gfCNCPoint4[4846] = {X 266.6262, Y 56.8093, Z -5.5000, A 0.000, B 0.000, C 0.000 }
gfCNCPoint4[4847] = {X 266.8456, Y 55.6367, Z -5.5000, A 0.000, B 0.000, C 0.000 }
gfCNCPoint4[4848] = {X 267.2076, Y 54.5000, Z -5.5000, A 0.000, B 0.000, C 0.000 }
gfCNCPoint4[4849] = {X 267.7067, Y 53.4164, Z -5.5000, A 0.000, B 0.000, C 0.000 }
gfCNCPoint4[4850] = {X 268.4728, Y 52.2132, Z -5.5000, A 0.000, B 0.000, C 0.000 }
gfCNCPoint4[4851] = {X 269.4075, Y 51.1357, Z -5.5000, A 0.000, B 0.000, C 0.000 }
gfCNCPoint4[4852] = {X 270.4903, Y 50.2072, Z -5.5000, A 0.000, B 0.000, C 0.000 }
gfCNCPoint4[4853] = {X 271.6979, Y 49.4479, Z -5.5000, A 0.000, B 0.000, C 0.000 }
gfCNCPoint4[4854] = {X 273.0039, Y 48.8744, Z -5.5000, A 0.000, B 0.000, C 0.000 }
gfCNCPoint4[4855] = {X 274.3800, Y 48.4989, Z -5.5000, A 0.000, B 0.000, C 0.000 }
gfCNCPoint4[4856] = {X 275.3020, Y 48.3648, Z -5.5000, A 0.000, B 0.000, C 0.000 }
gfCNCPoint4[4857] = {X 276.2327, Y 48.3200, Z -5.5000, A 0.000, B 0.000, C 0.000 }
gfCNCPoint4[4858] = {X 281.0411, Y 48.3200, Z -5.5000, A 0.000, B 0.000, C 0.000 }
gfCNCPoint4[4859] = {X 280.4347, Y 47.5134, Z -5.5000, A 0.000, B 0.000, C 0.000 }
gfCNCPoint4[4860] = {X 280.0072, Y 46.5992, Z -5.5000, A 0.000, B 0.000, C 0.000 }
gfCNCPoint4[4861] = {X 279.7768, Y 45.6167, Z -5.5000, A 0.000, B 0.000, C 0.000 }
gfCNCPoint4[4862] = {X 279.7488, Y 45.3288, Z -5.5000, A 0.000, B 0.000, C 0.000 }
gfCNCPoint4[4863] = {X 279.7378, Y 45.0398, Z -5.5000, A 0.000, B 0.000, C 0.000 }
gfCNCPoint4[4864] = {X 279.7377, Y 44.2045, Z -5.5000, A 0.000, B 0.000, C 0.000 }
gfCNCPoint4[4865] = {X 279.8418, Y 43.2208, Z -5.5000, A 0.000, B 0.000, C 0.000 }
gfCNCPoint4[4866] = {X 280.1403, Y 42.2777, Z -5.5000, A 0.000, B 0.000, C 0.000 }
gfCNCPoint4[4867] = {X 280.6212, Y 41.4133, Z -5.5000, A 0.000, B 0.000, C 0.000 }
gfCNCPoint4[4868] = {X 281.2650, Y 40.6623, Z -5.5000, A 0.000, B 0.000, C 0.000 }
gfCNCPoint4[4869] = {X 281.2646, Y 16.5236, Z -5.5000, A 0.000, B 0.000, C 0.000 }
gfCNCPoint4[4870] = {X 280.6237, Y 15.7821, Z -5.5000, A 0.000, B 0.000, C 0.000 }
gfCNCPoint4[4871] = {X 280.1439, Y 14.9274, Z -5.5000, A 0.000, B 0.000, C 0.000 }
gfCNCPoint4[4872] = {X 279.8446, Y 13.9941, Z -5.5000, A 0.000, B 0.000, C 0.000 }
gfCNCPoint4[4873] = {X 279.7378, Y 13.0198, Z -5.5000, A 0.000, B 0.000, C 0.000 }
gfCNCPoint4[4874] = {X 279.7377, Y 12.1868, Z -5.5000, A 0.000, B 0.000, C 0.000 }
gfCNCPoint4[4875] = {X 279.8242, Y 11.2717, Z -5.5000, A 0.000, B 0.000, C 0.000 }
gfCNCPoint4[4876] = {X 280.0809, Y 10.3891, Z -5.5000, A 0.000, B 0.000, C 0.000 }
gfCNCPoint4[4877] = {X 280.5256, Y 9.5280, Z -5.5000, A 0.000, B 0.000, C 0.000 }
gfCNCPoint4[4878] = {X 281.1317, Y 8.7718, Z -5.5000, A 0.000, B 0.000, C 0.000 }
gfCNCPoint4[4879] = {X 281.8753, Y 8.1503, Z -5.5000, A 0.000, B 0.000, C 0.000 }
gfCNCPoint4[4880] = {X 282.7270, Y 7.6879, Z -5.5000, A 0.000, B 0.000, C 0.000 }
gfCNCPoint4[4881] = {X 283.6533, Y 7.4030, Z -5.5000, A 0.000, B 0.000, C 0.000 }
gfCNCPoint4[4882] = {X 284.6177, Y 7.3068, Z -5.5000, A 0.000, B 0.000, C 0.000 }
gfCNCPoint4[4883] = {X 291.0611, Y 7.3068, Z -5.5000, A 0.000, B 0.000, C 0.000 }
gfCNCPoint4[4884] = {X 292.0255, Y 7.4030, Z -5.5000, A 0.000, B 0.000, C 0.000 }
gfCNCPoint4[4885] = {X 292.9518, Y 7.6879, Z -5.5000, A 0.000, B 0.000, C 0.000 }
gfCNCPoint4[4886] = {X 293.8035, Y 8.1503, Z -5.5000, A 0.000, B 0.000, C 0.000 }
gfCNCPoint4[4887] = {X 294.5471, Y 8.7718, Z -5.5000, A 0.000, B 0.000, C 0.000 }
gfCNCPoint4[4888] = {X 295.1532, Y 9.5280, Z -5.5000, A 0.000, B 0.000, C 0.000 }
gfCNCPoint4[4889] = {X 295.5979, Y 10.3891, Z -5.5000, A 0.000, B 0.000, C 0.000 }
gfCNCPoint4[4890] = {X 295.8044, Y 11.0397, Z -5.5000, A 0.000, B 0.000, C 0.000 }
gfCNCPoint4[4891] = {X 295.9180, Y 11.7127, Z -5.5000, A 0.000, B 0.000, C 0.000 }
gfCNCPoint4[4892] = {X 295.9354, Y 11.9495, Z -5.5000, A 0.000, B 0.000, C 0.000 }
gfCNCPoint4[4893] = {X 295.9411, Y 12.1868, Z -5.5000, A 0.000, B 0.000, C 0.000 }
gfCNCPoint4[4894] = {X 295.9409, Y 13.0237, Z -5.5000, A 0.000, B 0.000, C 0.000 }
gfCNCPoint4[4895] = {X 295.9342, Y 13.2382, Z -5.5000, A 0.000, B 0.000, C 0.000 }
gfCNCPoint4[4896] = {X 295.9180, Y 13.4521, Z -5.5000, A 0.000, B 0.000, C 0.000 }
gfCNCPoint4[4897] = {X 298.3067, Y 13.6853, Z -5.5000, A 0.000, B 0.000, C 0.000 }
gfCNCPoint4[4898] = {X 298.1361, Y 14.6935, Z -5.5000, A 0.000, B 0.000, C 0.000 }
gfCNCPoint4[4899] = {X 297.8260, Y 15.6678, Z -5.5000, A 0.000, B 0.000, C 0.000 }
gfCNCPoint4[4900] = {X 297.3824, Y 16.5891, Z -5.5000, A 0.000, B 0.000, C 0.000 }
gfCNCPoint4[4901] = {X 296.8141, Y 17.4392, Z -5.5000, A 0.000, B 0.000, C 0.000 }
gfCNCPoint4[4902] = {X 296.8144, Y 19.2365, Z -5.5000, A 0.000, B 0.000, C 0.000 }
gfCNCPoint4[4903] = {X 299.7989, Y 19.2365, Z -5.5000, A 0.000, B 0.000, C 0.000 }
gfCNCPoint4[4904] = {X 299.7990, Y 17.4388, Z -5.5000, A 0.000, B 0.000, C 0.000 }
gfCNCPoint4[4905] = {X 299.2308, Y 16.5888, Z -5.5000, A 0.000, B 0.000, C 0.000 }
gfCNCPoint4[4906] = {X 298.7873, Y 15.6676, Z -5.5000, A 0.000, B 0.000, C 0.000 }
gfCNCPoint4[4907] = {X 298.4772, Y 14.6934, Z -5.5000, A 0.000, B 0.000, C 0.000 }
gfCNCPoint4[4908] = {X 298.3067, Y 13.6853, Z -5.5000, A 0.000, B 0.000, C 0.000 }
gfCNCPoint4[4909] = {X 295.9180, Y 13.4521, Z -5.5000, A 0.000, B 0.000, C 0.000 }
gfCNCPoint4[4910] = {X 295.7560, Y 14.3094, Z -5.5000, A 0.000, B 0.000, C 0.000 }
gfCNCPoint4[4911] = {X 295.4439, Y 15.1241, Z -5.5000, A 0.000, B 0.000, C 0.000 }
gfCNCPoint4[4912] = {X 294.9917, Y 15.8702, Z -5.5000, A 0.000, B 0.000, C 0.000 }
gfCNCPoint4[4913] = {X 294.4139, Y 16.5239, Z -5.5000, A 0.000, B 0.000, C 0.000 }
gfCNCPoint4[4914] = {X 294.4148, Y 21.6365, Z -5.5000, A 0.000, B 0.000, C 0.000 }
gfCNCPoint4[4915] = {X 302.1988, Y 21.6365, Z -5.5000, A 0.000, B 0.000, C 0.000 }
gfCNCPoint4[4916] = {X 302.1991, Y 16.5235, Z -5.5000, A 0.000, B 0.000, C 0.000 }
gfCNCPoint4[4917] = {X 301.6214, Y 15.8699, Z -5.5000, A 0.000, B 0.000, C 0.000 }
gfCNCPoint4[4918] = {X 301.1694, Y 15.1239, Z -5.5000, A 0.000, B 0.000, C 0.000 }
gfCNCPoint4[4919] = {X 300.8573, Y 14.3093, Z -5.5000, A 0.000, B 0.000, C 0.000 }
gfCNCPoint4[4920] = {X 300.6953, Y 13.4521, Z -5.5000, A 0.000, B 0.000, C 0.000 }
gfCNCPoint4[4921] = {X 300.6791, Y 13.2371, Z -5.5000, A 0.000, B 0.000, C 0.000 }
gfCNCPoint4[4922] = {X 300.6724, Y 13.0215, Z -5.5000, A 0.000, B 0.000, C 0.000 }
gfCNCPoint4[4923] = {X 300.6723, Y 12.1868, Z -5.5000, A 0.000, B 0.000, C 0.000 }
gfCNCPoint4[4924] = {X 300.6780, Y 11.9495, Z -5.5000, A 0.000, B 0.000, C 0.000 }
gfCNCPoint4[4925] = {X 300.6953, Y 11.7127, Z -5.5000, A 0.000, B 0.000, C 0.000 }
gfCNCPoint4[4926] = {X 300.8090, Y 11.0397, Z -5.5000, A 0.000, B 0.000, C 0.000 }
gfCNCPoint4[4927] = {X 301.0155, Y 10.3891, Z -5.5000, A 0.000, B 0.000, C 0.000 }
gfCNCPoint4[4928] = {X 301.4602, Y 9.5280, Z -5.5000, A 0.000, B 0.000, C 0.000 }
gfCNCPoint4[4929] = {X 302.0663, Y 8.7718, Z -5.5000, A 0.000, B 0.000, C 0.000 }
gfCNCPoint4[4930] = {X 302.8099, Y 8.1503, Z -5.5000, A 0.000, B 0.000, C 0.000 }
gfCNCPoint4[4931] = {X 303.6616, Y 7.6879, Z -5.5000, A 0.000, B 0.000, C 0.000 }
gfCNCPoint4[4932] = {X 304.5879, Y 7.4030, Z -5.5000, A 0.000, B 0.000, C 0.000 }
gfCNCPoint4[4933] = {X 305.5523, Y 7.3068, Z -5.5000, A 0.000, B 0.000, C 0.000 }
gfCNCPoint4[4934] = {X 311.9957, Y 7.3068, Z -5.5000, A 0.000, B 0.000, C 0.000 }
gfCNCPoint4[4935] = {X 312.9478, Y 7.4006, Z -5.5000, A 0.000, B 0.000, C 0.000 }
gfCNCPoint4[4936] = {X 313.8632, Y 7.6783, Z -5.5000, A 0.000, B 0.000, C 0.000 }
gfCNCPoint4[4937] = {X 314.7069, Y 8.1292, Z -5.5000, A 0.000, B 0.000, C 0.000 }
gfCNCPoint4[4938] = {X 315.4464, Y 8.7361, Z -5.5000, A 0.000, B 0.000, C 0.000 }
gfCNCPoint4[4939] = {X 316.0533, Y 9.4756, Z -5.5000, A 0.000, B 0.000, C 0.000 }
gfCNCPoint4[4940] = {X 316.5043, Y 10.3193, Z -5.5000, A 0.000, B 0.000, C 0.000 }
gfCNCPoint4[4941] = {X 316.7820, Y 11.2348, Z -5.5000, A 0.000, B 0.000, C 0.000 }
gfCNCPoint4[4942] = {X 316.8757, Y 12.1868, Z -5.5000, A 0.000, B 0.000, C 0.000 }
gfCNCPoint4[4943] = {X 316.8755, Y 13.0237, Z -5.5000, A 0.000, B 0.000, C 0.000 }
gfCNCPoint4[4944] = {X 316.7682, Y 13.9967, Z -5.5000, A 0.000, B 0.000, C 0.000 }
gfCNCPoint4[4945] = {X 316.4689, Y 14.9287, Z -5.5000, A 0.000, B 0.000, C 0.000 }
gfCNCPoint4[4946] = {X 315.9895, Y 15.7823, Z -5.5000, A 0.000, B 0.000, C 0.000 }
gfCNCPoint4[4947] = {X 315.3495, Y 16.5229, Z -5.5000, A 0.000, B 0.000, C 0.000 }
gfCNCPoint4[4948] = {X 315.3484, Y 40.6628, Z -5.5000, A 0.000, B 0.000, C 0.000 }
gfCNCPoint4[4949] = {X 315.9894, Y 41.4043, Z -5.5000, A 0.000, B 0.000, C 0.000 }
gfCNCPoint4[4950] = {X 316.4692, Y 42.2589, Z -5.5000, A 0.000, B 0.000, C 0.000 }
gfCNCPoint4[4951] = {X 316.7687, Y 43.1922, Z -5.5000, A 0.000, B 0.000, C 0.000 }
gfCNCPoint4[4952] = {X 316.8755, Y 44.1664, Z -5.5000, A 0.000, B 0.000, C 0.000 }
gfCNCPoint4[4953] = {X 316.8757, Y 45.0000, Z -5.5000, A 0.000, B 0.000, C 0.000 }
gfCNCPoint4[4954] = {X 316.8749, Y 45.0899, Z -5.5000, A 0.000, B 0.000, C 0.000 }
gfCNCPoint4[4955] = {X 316.8724, Y 45.1799, Z -5.5000, A 0.000, B 0.000, C 0.000 }
gfCNCPoint4[4956] = {X 316.8594, Y 45.3987, Z -5.5000, A 0.000, B 0.000, C 0.000 }
gfCNCPoint4[4957] = {X 316.8366, Y 45.6167, Z -5.5000, A 0.000, B 0.000, C 0.000 }
gfCNCPoint4[4958] = {X 316.6062, Y 46.5992, Z -5.5000, A 0.000, B 0.000, C 0.000 }
gfCNCPoint4[4959] = {X 316.1787, Y 47.5134, Z -5.5000, A 0.000, B 0.000, C 0.000 }
gfCNCPoint4[4960] = {X 315.5723, Y 48.3200, Z -5.5000, A 0.000, B 0.000, C 0.000 }
gfCNCPoint4[4961] = {X 315.2205, Y 47.9934, Z -5.5000, A 0.000, B 0.000, C 0.000 }
gfCNCPoint4[4962] = {X 314.5413, Y 48.5889, Z -5.5000, A 0.000, B 0.000, C 0.000 }
gfCNCPoint4[4963] = {X 313.7548, Y 49.0331, Z -5.5000, A 0.000, B 0.000, C 0.000 }
gfCNCPoint4[4964] = {X 312.8942, Y 49.3073, Z -5.5000, A 0.000, B 0.000, C 0.000 }
gfCNCPoint4[4965] = {X 311.9957, Y 49.4000, Z -5.5000, A 0.000, B 0.000, C 0.000 }
gfCNCPoint4[4966] = {X 305.5523, Y 49.4000, Z -5.5000, A 0.000, B 0.000, C 0.000 }
gfCNCPoint4[4967] = {X 304.5732, Y 49.2897, Z -5.5000, A 0.000, B 0.000, C 0.000 }
gfCNCPoint4[4968] = {X 303.6432, Y 48.9643, Z -5.5000, A 0.000, B 0.000, C 0.000 }
gfCNCPoint4[4969] = {X 302.8089, Y 48.4400, Z -5.5000, A 0.000, B 0.000, C 0.000 }
gfCNCPoint4[4970] = {X 302.1122, Y 47.7433, Z -5.5000, A 0.000, B 0.000, C 0.000 }
gfCNCPoint4[4971] = {X 301.5880, Y 46.9091, Z -5.5000, A 0.000, B 0.000, C 0.000 }
gfCNCPoint4[4972] = {X 301.2626, Y 45.9791, Z -5.5000, A 0.000, B 0.000, C 0.000 }
gfCNCPoint4[4973] = {X 301.1523, Y 45.0000, Z -5.5000, A 0.000, B 0.000, C 0.000 }
gfCNCPoint4[4974] = {X 301.1524, Y 44.1994, Z -5.5000, A 0.000, B 0.000, C 0.000 }
gfCNCPoint4[4975] = {X 301.2698, Y 43.2559, Z -5.5000, A 0.000, B 0.000, C 0.000 }
gfCNCPoint4[4976] = {X 301.5727, Y 42.3547, Z -5.5000, A 0.000, B 0.000, C 0.000 }
gfCNCPoint4[4977] = {X 302.0489, Y 41.5318, Z -5.5000, A 0.000, B 0.000, C 0.000 }
gfCNCPoint4[4978] = {X 302.6794, Y 40.8202, Z -5.5000, A 0.000, B 0.000, C 0.000 }
gfCNCPoint4[4979] = {X 302.6794, Y 34.1143, Z -5.5000, A 0.000, B 0.000, C 0.000 }
gfCNCPoint4[4980] = {X 293.9347, Y 34.1143, Z -5.5000, A 0.000, B 0.000, C 0.000 }
gfCNCPoint4[4981] = {X 293.9340, Y 40.8658, Z -5.5000, A 0.000, B 0.000, C 0.000 }
gfCNCPoint4[4982] = {X 294.5740, Y 41.5608, Z -5.5000, A 0.000, B 0.000, C 0.000 }
gfCNCPoint4[4983] = {X 295.0547, Y 42.3742, Z -5.5000, A 0.000, B 0.000, C 0.000 }
gfCNCPoint4[4984] = {X 295.3548, Y 43.2701, Z -5.5000, A 0.000, B 0.000, C 0.000 }
gfCNCPoint4[4985] = {X 295.4611, Y 44.2089, Z -5.5000, A 0.000, B 0.000, C 0.000 }
gfCNCPoint4[4986] = {X 295.4611, Y 45.0000, Z -5.5000, A 0.000, B 0.000, C 0.000 }
gfCNCPoint4[4987] = {X 295.3508, Y 45.9791, Z -5.5000, A 0.000, B 0.000, C 0.000 }
gfCNCPoint4[4988] = {X 295.0254, Y 46.9091, Z -5.5000, A 0.000, B 0.000, C 0.000 }
gfCNCPoint4[4989] = {X 294.5012, Y 47.7434, Z -5.5000, A 0.000, B 0.000, C 0.000 }
gfCNCPoint4[4990] = {X 293.8045, Y 48.4401, Z -5.5000, A 0.000, B 0.000, C 0.000 }
gfCNCPoint4[4991] = {X 292.9702, Y 48.9643, Z -5.5000, A 0.000, B 0.000, C 0.000 }
gfCNCPoint4[4992] = {X 292.0402, Y 49.2897, Z -5.5000, A 0.000, B 0.000, C 0.000 }
gfCNCPoint4[4993] = {X 291.0611, Y 49.4000, Z -5.5000, A 0.000, B 0.000, C 0.000 }
gfCNCPoint4[4994] = {X 284.6177, Y 49.4000, Z -5.5000, A 0.000, B 0.000, C 0.000 }
gfCNCPoint4[4995] = {X 283.6386, Y 49.2897, Z -5.5000, A 0.000, B 0.000, C 0.000 }
gfCNCPoint4[4996] = {X 282.7086, Y 48.9643, Z -5.5000, A 0.000, B 0.000, C 0.000 }
gfCNCPoint4[4997] = {X 281.8743, Y 48.4400, Z -5.5000, A 0.000, B 0.000, C 0.000 }
gfCNCPoint4[4998] = {X 281.1776, Y 47.7433, Z -5.5000, A 0.000, B 0.000, C 0.000 }
gfCNCPoint4[4999] = {X 280.6534, Y 46.9091, Z -5.5000, A 0.000, B 0.000, C 0.000 }
gfCNCPoint4[5000] = {X 280.3280, Y 45.9791, Z -5.5000, A 0.000, B 0.000, C 0.000 }
gfCNCPoint4[5001] = {X 280.2177, Y 45.0000, Z -5.5000, A 0.000, B 0.000, C 0.000 }
gfCNCPoint4[5002] = {X 280.2177, Y 44.2069, Z -5.5000, A 0.000, B 0.000, C 0.000 }
gfCNCPoint4[5003] = {X 280.3222, Y 43.2698, Z -5.5000, A 0.000, B 0.000, C 0.000 }
gfCNCPoint4[5004] = {X 280.6220, Y 42.3758, Z -5.5000, A 0.000, B 0.000, C 0.000 }
gfCNCPoint4[5005] = {X 281.1034, Y 41.5651, Z -5.5000, A 0.000, B 0.000, C 0.000 }
gfCNCPoint4[5006] = {X 281.7450, Y 40.8741, Z -5.5000, A 0.000, B 0.000, C 0.000 }
gfCNCPoint4[5007] = {X 281.7446, Y 16.3105, Z -5.5000, A 0.000, B 0.000, C 0.000 }
gfCNCPoint4[5008] = {X 281.1002, Y 15.6214, Z -5.5000, A 0.000, B 0.000, C 0.000 }
gfCNCPoint4[5009] = {X 280.6176, Y 14.8108, Z -5.5000, A 0.000, B 0.000, C 0.000 }
gfCNCPoint4[5010] = {X 280.3188, Y 13.9159, Z -5.5000, A 0.000, B 0.000, C 0.000 }
gfCNCPoint4[5011] = {X 280.2177, Y 12.9780, Z -5.5000, A 0.000, B 0.000, C 0.000 }
gfCNCPoint4[5012] = {X 280.2177, Y 12.1868, Z -5.5000, A 0.000, B 0.000, C 0.000 }
gfCNCPoint4[5013] = {X 280.3280, Y 11.2077, Z -5.5000, A 0.000, B 0.000, C 0.000 }
gfCNCPoint4[5014] = {X 280.6534, Y 10.2777, Z -5.5000, A 0.000, B 0.000, C 0.000 }
gfCNCPoint4[5015] = {X 281.1776, Y 9.4435, Z -5.5000, A 0.000, B 0.000, C 0.000 }
gfCNCPoint4[5016] = {X 281.8743, Y 8.7468, Z -5.5000, A 0.000, B 0.000, C 0.000 }
gfCNCPoint4[5017] = {X 282.7086, Y 8.2226, Z -5.5000, A 0.000, B 0.000, C 0.000 }
gfCNCPoint4[5018] = {X 283.6386, Y 7.8971, Z -5.5000, A 0.000, B 0.000, C 0.000 }
gfCNCPoint4[5019] = {X 284.6177, Y 7.7868, Z -5.5000, A 0.000, B 0.000, C 0.000 }
gfCNCPoint4[5020] = {X 291.0611, Y 7.7868, Z -5.5000, A 0.000, B 0.000, C 0.000 }
gfCNCPoint4[5021] = {X 292.0402, Y 7.8971, Z -5.5000, A 0.000, B 0.000, C 0.000 }
gfCNCPoint4[5022] = {X 292.9702, Y 8.2226, Z -5.5000, A 0.000, B 0.000, C 0.000 }
gfCNCPoint4[5023] = {X 293.8045, Y 8.7468, Z -5.5000, A 0.000, B 0.000, C 0.000 }
gfCNCPoint4[5024] = {X 294.5012, Y 9.4435, Z -5.5000, A 0.000, B 0.000, C 0.000 }
gfCNCPoint4[5025] = {X 295.0254, Y 10.2777, Z -5.5000, A 0.000, B 0.000, C 0.000 }
gfCNCPoint4[5026] = {X 295.3508, Y 11.2077, Z -5.5000, A 0.000, B 0.000, C 0.000 }
gfCNCPoint4[5027] = {X 295.4611, Y 12.1868, Z -5.5000, A 0.000, B 0.000, C 0.000 }
gfCNCPoint4[5028] = {X 295.4609, Y 13.0233, Z -5.5000, A 0.000, B 0.000, C 0.000 }
gfCNCPoint4[5029] = {X 295.3526, Y 13.9493, Z -5.5000, A 0.000, B 0.000, C 0.000 }
gfCNCPoint4[5030] = {X 295.0517, Y 14.8316, Z -5.5000, A 0.000, B 0.000, C 0.000 }
gfCNCPoint4[5031] = {X 294.5716, Y 15.6307, Z -5.5000, A 0.000, B 0.000, C 0.000 }
gfCNCPoint4[5032] = {X 293.9339, Y 16.3108, Z -5.5000, A 0.000, B 0.000, C 0.000 }
gfCNCPoint4[5033] = {X 293.9349, Y 22.1165, Z -5.5000, A 0.000, B 0.000, C 0.000 }
gfCNCPoint4[5034] = {X 302.6787, Y 22.1165, Z -5.5000, A 0.000, B 0.000, C 0.000 }
gfCNCPoint4[5035] = {X 302.6791, Y 16.3104, Z -5.5000, A 0.000, B 0.000, C 0.000 }
gfCNCPoint4[5036] = {X 302.0348, Y 15.6214, Z -5.5000, A 0.000, B 0.000, C 0.000 }
gfCNCPoint4[5037] = {X 301.5521, Y 14.8108, Z -5.5000, A 0.000, B 0.000, C 0.000 }
gfCNCPoint4[5038] = {X 301.2534, Y 13.9159, Z -5.5000, A 0.000, B 0.000, C 0.000 }
gfCNCPoint4[5039] = {X 301.1523, Y 12.9779, Z -5.5000, A 0.000, B 0.000, C 0.000 }
gfCNCPoint4[5040] = {X 301.1523, Y 12.1868, Z -5.5000, A 0.000, B 0.000, C 0.000 }
gfCNCPoint4[5041] = {X 301.2626, Y 11.2077, Z -5.5000, A 0.000, B 0.000, C 0.000 }
gfCNCPoint4[5042] = {X 301.5880, Y 10.2777, Z -5.5000, A 0.000, B 0.000, C 0.000 }
gfCNCPoint4[5043] = {X 302.1122, Y 9.4435, Z -5.5000, A 0.000, B 0.000, C 0.000 }
gfCNCPoint4[5044] = {X 302.8089, Y 8.7468, Z -5.5000, A 0.000, B 0.000, C 0.000 }
gfCNCPoint4[5045] = {X 303.6432, Y 8.2226, Z -5.5000, A 0.000, B 0.000, C 0.000 }
gfCNCPoint4[5046] = {X 304.5732, Y 7.8971, Z -5.5000, A 0.000, B 0.000, C 0.000 }
gfCNCPoint4[5047] = {X 305.5523, Y 7.7868, Z -5.5000, A 0.000, B 0.000, C 0.000 }
gfCNCPoint4[5048] = {X 311.9957, Y 7.7868, Z -5.5000, A 0.000, B 0.000, C 0.000 }
gfCNCPoint4[5049] = {X 312.9748, Y 7.8971, Z -5.5000, A 0.000, B 0.000, C 0.000 }
gfCNCPoint4[5050] = {X 313.9048, Y 8.2226, Z -5.5000, A 0.000, B 0.000, C 0.000 }
gfCNCPoint4[5051] = {X 314.7391, Y 8.7468, Z -5.5000, A 0.000, B 0.000, C 0.000 }
gfCNCPoint4[5052] = {X 315.4358, Y 9.4435, Z -5.5000, A 0.000, B 0.000, C 0.000 }
gfCNCPoint4[5053] = {X 315.9600, Y 10.2777, Z -5.5000, A 0.000, B 0.000, C 0.000 }
gfCNCPoint4[5054] = {X 316.2854, Y 11.2077, Z -5.5000, A 0.000, B 0.000, C 0.000 }
gfCNCPoint4[5055] = {X 316.3957, Y 12.1868, Z -5.5000, A 0.000, B 0.000, C 0.000 }
gfCNCPoint4[5056] = {X 316.3955, Y 13.0233, Z -5.5000, A 0.000, B 0.000, C 0.000 }
gfCNCPoint4[5057] = {X 316.2873, Y 13.9489, Z -5.5000, A 0.000, B 0.000, C 0.000 }
gfCNCPoint4[5058] = {X 315.9865, Y 14.8310, Z -5.5000, A 0.000, B 0.000, C 0.000 }
gfCNCPoint4[5059] = {X 315.5068, Y 15.6299, Z -5.5000, A 0.000, B 0.000, C 0.000 }
gfCNCPoint4[5060] = {X 314.8695, Y 16.3099, Z -5.5000, A 0.000, B 0.000, C 0.000 }
gfCNCPoint4[5061] = {X 314.8684, Y 40.8760, Z -5.5000, A 0.000, B 0.000, C 0.000 }
gfCNCPoint4[5062] = {X 315.5129, Y 41.5651, Z -5.5000, A 0.000, B 0.000, C 0.000 }
gfCNCPoint4[5063] = {X 315.9957, Y 42.3758, Z -5.5000, A 0.000, B 0.000, C 0.000 }
gfCNCPoint4[5064] = {X 316.2946, Y 43.2708, Z -5.5000, A 0.000, B 0.000, C 0.000 }
gfCNCPoint4[5065] = {X 316.3957, Y 44.2089, Z -5.5000, A 0.000, B 0.000, C 0.000 }
gfCNCPoint4[5066] = {X 316.3957, Y 45.0000, Z -5.5000, A 0.000, B 0.000, C 0.000 }
gfCNCPoint4[5067] = {X 316.3190, Y 45.8182, Z -5.5000, A 0.000, B 0.000, C 0.000 }
gfCNCPoint4[5068] = {X 316.0914, Y 46.6079, Z -5.5000, A 0.000, B 0.000, C 0.000 }
gfCNCPoint4[5069] = {X 315.7209, Y 47.3415, Z -5.5000, A 0.000, B 0.000, C 0.000 }
gfCNCPoint4[5070] = {X 315.2205, Y 47.9934, Z -5.5000, A 0.000, B 0.000, C 0.000 }
gfCNCPoint4[5071] = {X 315.5723, Y 48.3200, Z -5.5000, A 0.000, B 0.000, C 0.000 }
gfCNCPoint4[5072] = {X 324.3107, Y 48.3200, Z -5.5000, A 0.000, B 0.000, C 0.000 }
gfCNCPoint4[5073] = {X 325.5555, Y 48.4004, Z -5.5000, A 0.000, B 0.000, C 0.000 }
gfCNCPoint4[5074] = {X 326.7797, Y 48.6402, Z -5.5000, A 0.000, B 0.000, C 0.000 }
gfCNCPoint4[5075] = {X 325.5882, Y 48.0963, Z -5.5000, A 0.000, B 0.000, C 0.000 }
gfCNCPoint4[5076] = {X 324.4810, Y 47.3966, Z -5.5000, A 0.000, B 0.000, C 0.000 }
gfCNCPoint4[5077] = {X 323.4784, Y 46.5538, Z -5.5000, A 0.000, B 0.000, C 0.000 }
gfCNCPoint4[5078] = {X 322.8382, Y 45.9295, Z -5.5000, A 0.000, B 0.000, C 0.000 }
gfCNCPoint4[5079] = {X 322.2180, Y 45.2650, Z -5.5000, A 0.000, B 0.000, C 0.000 }
gfCNCPoint4[5080] = {X 321.6628, Y 44.5452, Z -5.5000, A 0.000, B 0.000, C 0.000 }
gfCNCPoint4[5081] = {X 323.6300, Y 43.1703, Z -5.5000, A 0.000, B 0.000, C 0.000 }
gfCNCPoint4[5082] = {X 323.0063, Y 42.0918, Z -5.5000, A 0.000, B 0.000, C 0.000 }
gfCNCPoint4[5083] = {X 322.5757, Y 40.9227, Z -5.5000, A 0.000, B 0.000, C 0.000 }
gfCNCPoint4[5084] = {X 322.3506, Y 39.6973, Z -5.5000, A 0.000, B 0.000, C 0.000 }
gfCNCPoint4[5085] = {X 322.3379, Y 38.4514, Z -5.5000, A 0.000, B 0.000, C 0.000 }
gfCNCPoint4[5086] = {X 322.5377, Y 37.2217, Z -5.5000, A 0.000, B 0.000, C 0.000 }
gfCNCPoint4[5087] = {X 322.9443, Y 36.0440, Z -5.5000, A 0.000, B 0.000, C 0.000 }
gfCNCPoint4[5088] = {X 323.5458, Y 34.9529, Z -5.5000, A 0.000, B 0.000, C 0.000 }
gfCNCPoint4[5089] = {X 327.7840, Y 28.6158, Z -5.5000, A 0.000, B 0.000, C 0.000 }
gfCNCPoint4[5090] = {X 328.5200, Y 27.6906, Z -5.5000, A 0.000, B 0.000, C 0.000 }
gfCNCPoint4[5091] = {X 329.3960, Y 26.8968, Z -5.5000, A 0.000, B 0.000, C 0.000 }
gfCNCPoint4[5092] = {X 330.3889, Y 26.2552, Z -5.5000, A 0.000, B 0.000, C 0.000 }
gfCNCPoint4[5093] = {X 331.5063, Y 25.7713, Z -5.5000, A 0.000, B 0.000, C 0.000 }
gfCNCPoint4[5094] = {X 332.6887, Y 25.4804, Z -5.5000, A 0.000, B 0.000, C 0.000 }
gfCNCPoint4[5095] = {X 333.9031, Y 25.3907, Z -5.5000, A 0.000, B 0.000, C 0.000 }
gfCNCPoint4[5096] = {X 335.1154, Y 25.5046, Z -5.5000, A 0.000, B 0.000, C 0.000 }
gfCNCPoint4[5097] = {X 336.2918, Y 25.8191, Z -5.5000, A 0.000, B 0.000, C 0.000 }
gfCNCPoint4[5098] = {X 337.3993, Y 26.3252, Z -5.5000, A 0.000, B 0.000, C 0.000 }
gfCNCPoint4[5099] = {X 338.1754, Y 26.8291, Z -5.5000, A 0.000, B 0.000, C 0.000 }
gfCNCPoint4[5100] = {X 338.8812, Y 27.4275, Z -5.5000, A 0.000, B 0.000, C 0.000 }
gfCNCPoint4[5101] = {X 339.5029, Y 28.0268, Z -5.5000, A 0.000, B 0.000, C 0.000 }
gfCNCPoint4[5102] = {X 340.3307, Y 28.9967, Z -5.5000, A 0.000, B 0.000, C 0.000 }
gfCNCPoint4[5103] = {X 340.9766, Y 30.0961, Z -5.5000, A 0.000, B 0.000, C 0.000 }
gfCNCPoint4[5104] = {X 341.4207, Y 31.2913, Z -5.5000, A 0.000, B 0.000, C 0.000 }
gfCNCPoint4[5105] = {X 341.6495, Y 32.5458, Z -5.5000, A 0.000, B 0.000, C 0.000 }
gfCNCPoint4[5106] = {X 341.8492, Y 32.7096, Z -5.5000, A 0.000, B 0.000, C 0.000 }
gfCNCPoint4[5107] = {X 342.0509, Y 32.8710, Z -5.5000, A 0.000, B 0.000, C 0.000 }
gfCNCPoint4[5108] = {X 342.9928, Y 33.4854, Z -5.5000, A 0.000, B 0.000, C 0.000 }
gfCNCPoint4[5109] = {X 344.0146, Y 33.9553, Z -5.5000, A 0.000, B 0.000, C 0.000 }
gfCNCPoint4[5110] = {X 345.0942, Y 34.2706, Z -5.5000, A 0.000, B 0.000, C 0.000 }
gfCNCPoint4[5111] = {X 346.2082, Y 34.4244, Z -5.5000, A 0.000, B 0.000, C 0.000 }
gfCNCPoint4[5112] = {X 347.3328, Y 34.4134, Z -5.5000, A 0.000, B 0.000, C 0.000 }
gfCNCPoint4[5113] = {X 348.3024, Y 34.2880, Z -5.5000, A 0.000, B 0.000, C 0.000 }
gfCNCPoint4[5114] = {X 349.2382, Y 34.0050, Z -5.5000, A 0.000, B 0.000, C 0.000 }
gfCNCPoint4[5115] = {X 350.1149, Y 33.5723, Z -5.5000, A 0.000, B 0.000, C 0.000 }
gfCNCPoint4[5116] = {X 350.9086, Y 33.0016, Z -5.5000, A 0.000, B 0.000, C 0.000 }
gfCNCPoint4[5117] = {X 351.7848, Y 32.1504, Z -5.5000, A 0.000, B 0.000, C 0.000 }
gfCNCPoint4[5118] = {X 352.5433, Y 31.1929, Z -5.5000, A 0.000, B 0.000, C 0.000 }
gfCNCPoint4[5119] = {X 353.1713, Y 30.1451, Z -5.5000, A 0.000, B 0.000, C 0.000 }
gfCNCPoint4[5120] = {X 353.6581, Y 29.0247, Z -5.5000, A 0.000, B 0.000, C 0.000 }
gfCNCPoint4[5121] = {X 353.9955, Y 27.8507, Z -5.5000, A 0.000, B 0.000, C 0.000 }
gfCNCPoint4[5122] = {X 354.2230, Y 26.4400, Z -5.5000, A 0.000, B 0.000, C 0.000 }
gfCNCPoint4[5123] = {X 354.3150, Y 25.0140, Z -5.5000, A 0.000, B 0.000, C 0.000 }
gfCNCPoint4[5124] = {X 354.2708, Y 23.5858, Z -5.5000, A 0.000, B 0.000, C 0.000 }
gfCNCPoint4[5125] = {X 354.0907, Y 22.1682, Z -5.5000, A 0.000, B 0.000, C 0.000 }
gfCNCPoint4[5126] = {X 353.8258, Y 21.0252, Z -5.5000, A 0.000, B 0.000, C 0.000 }
gfCNCPoint4[5127] = {X 353.4125, Y 19.9271, Z -5.5000, A 0.000, B 0.000, C 0.000 }
gfCNCPoint4[5128] = {X 352.8580, Y 18.8931, Z -5.5000, A 0.000, B 0.000, C 0.000 }
gfCNCPoint4[5129] = {X 352.1719, Y 17.9412, Z -5.5000, A 0.000, B 0.000, C 0.000 }
gfCNCPoint4[5130] = {X 351.4220, Y 17.1682, Z -5.5000, A 0.000, B 0.000, C 0.000 }
gfCNCPoint4[5131] = {X 350.5495, Y 16.5369, Z -5.5000, A 0.000, B 0.000, C 0.000 }
gfCNCPoint4[5132] = {X 349.5808, Y 16.0663, Z -5.5000, A 0.000, B 0.000, C 0.000 }
gfCNCPoint4[5133] = {X 348.5452, Y 15.7708, Z -5.5000, A 0.000, B 0.000, C 0.000 }
gfCNCPoint4[5134] = {X 347.1588, Y 15.5996, Z -5.5000, A 0.000, B 0.000, C 0.000 }
gfCNCPoint4[5135] = {X 345.7620, Y 15.6153, Z -5.5000, A 0.000, B 0.000, C 0.000 }
gfCNCPoint4[5136] = {X 344.3798, Y 15.8177, Z -5.5000, A 0.000, B 0.000, C 0.000 }
gfCNCPoint4[5137] = {X 343.0371, Y 16.2031, Z -5.5000, A 0.000, B 0.000, C 0.000 }
gfCNCPoint4[5138] = {X 341.7580, Y 16.7647, Z -5.5000, A 0.000, B 0.000, C 0.000 }
gfCNCPoint4[5139] = {X 341.4303, Y 17.8594, Z -5.5000, A 0.000, B 0.000, C 0.000 }
gfCNCPoint4[5140] = {X 340.9353, Y 18.8894, Z -5.5000, A 0.000, B 0.000, C 0.000 }
gfCNCPoint4[5141] = {X 340.2853, Y 19.8292, Z -5.5000, A 0.000, B 0.000, C 0.000 }
gfCNCPoint4[5142] = {X 345.8671, Y 24.3770, Z -5.5000, A 0.000, B 0.000, C 0.000 }
gfCNCPoint4[5143] = {X 346.4656, Y 25.2129, Z -5.5000, A 0.000, B 0.000, C 0.000 }
gfCNCPoint4[5144] = {X 347.0033, Y 26.0891, Z -5.5000, A 0.000, B 0.000, C 0.000 }
gfCNCPoint4[5145] = {X 347.1058, Y 25.1827, Z -5.5000, A 0.000, B 0.000, C 0.000 }
gfCNCPoint4[5146] = {X 347.1016, Y 24.2705, Z -5.5000, A 0.000, B 0.000, C 0.000 }
gfCNCPoint4[5147] = {X 346.9906, Y 23.3651, Z -5.5000, A 0.000, B 0.000, C 0.000 }
gfCNCPoint4[5148] = {X 346.9492, Y 23.1616, Z -5.5000, A 0.000, B 0.000, C 0.000 }
gfCNCPoint4[5149] = {X 346.8829, Y 22.9649, Z -5.5000, A 0.000, B 0.000, C 0.000 }
gfCNCPoint4[5150] = {X 346.3963, Y 23.6862, Z -5.5000, A 0.000, B 0.000, C 0.000 }
gfCNCPoint4[5151] = {X 345.8671, Y 24.3770, Z -5.5000, A 0.000, B 0.000, C 0.000 }
gfCNCPoint4[5152] = {X 344.0065, Y 22.8611, Z -5.5000, A 0.000, B 0.000, C 0.000 }
gfCNCPoint4[5153] = {X 343.3271, Y 23.6263, Z -5.5000, A 0.000, B 0.000, C 0.000 }
gfCNCPoint4[5154] = {X 342.5854, Y 24.3313, Z -5.5000, A 0.000, B 0.000, C 0.000 }
gfCNCPoint4[5155] = {X 342.8589, Y 24.5950, Z -5.5000, A 0.000, B 0.000, C 0.000 }
gfCNCPoint4[5156] = {X 343.9806, Y 25.8609, Z -5.5000, A 0.000, B 0.000, C 0.000 }
gfCNCPoint4[5157] = {X 344.9145, Y 27.2710, Z -5.5000, A 0.000, B 0.000, C 0.000 }
gfCNCPoint4[5158] = {X 345.4663, Y 28.3741, Z -5.5000, A 0.000, B 0.000, C 0.000 }
gfCNCPoint4[5159] = {X 345.9028, Y 29.5278, Z -5.5000, A 0.000, B 0.000, C 0.000 }
gfCNCPoint4[5160] = {X 346.4603, Y 29.6308, Z -5.5000, A 0.000, B 0.000, C 0.000 }
gfCNCPoint4[5161] = {X 347.0272, Y 29.6217, Z -5.5000, A 0.000, B 0.000, C 0.000 }
gfCNCPoint4[5162] = {X 347.4362, Y 29.5565, Z -5.5000, A 0.000, B 0.000, C 0.000 }
gfCNCPoint4[5163] = {X 347.7945, Y 29.3488, Z -5.5000, A 0.000, B 0.000, C 0.000 }
gfCNCPoint4[5164] = {X 348.4747, Y 28.6292, Z -5.5000, A 0.000, B 0.000, C 0.000 }
gfCNCPoint4[5165] = {X 348.9852, Y 27.7809, Z -5.5000, A 0.000, B 0.000, C 0.000 }
gfCNCPoint4[5166] = {X 349.3025, Y 26.8429, Z -5.5000, A 0.000, B 0.000, C 0.000 }
gfCNCPoint4[5167] = {X 349.3368, Y 26.6707, Z -5.5000, A 0.000, B 0.000, C 0.000 }
gfCNCPoint4[5168] = {X 349.3683, Y 26.4979, Z -5.5000, A 0.000, B 0.000, C 0.000 }
gfCNCPoint4[5169] = {X 349.5017, Y 25.3238, Z -5.5000, A 0.000, B 0.000, C 0.000 }
gfCNCPoint4[5170] = {X 349.4982, Y 24.1421, Z -5.5000, A 0.000, B 0.000, C 0.000 }
gfCNCPoint4[5171] = {X 349.3578, Y 22.9688, Z -5.5000, A 0.000, B 0.000, C 0.000 }
gfCNCPoint4[5172] = {X 349.1799, Y 22.2566, Z -5.5000, A 0.000, B 0.000, C 0.000 }
gfCNCPoint4[5173] = {X 348.8773, Y 21.5878, Z -5.5000, A 0.000, B 0.000, C 0.000 }
gfCNCPoint4[5174] = {X 348.4596, Y 20.9841, Z -5.5000, A 0.000, B 0.000, C 0.000 }
gfCNCPoint4[5175] = {X 348.0926, Y 20.6604, Z -5.5000, A 0.000, B 0.000, C 0.000 }
gfCNCPoint4[5176] = {X 347.6362, Y 20.4840, Z -5.5000, A 0.000, B 0.000, C 0.000 }
gfCNCPoint4[5177] = {X 346.5778, Y 20.3833, Z -5.5000, A 0.000, B 0.000, C 0.000 }
gfCNCPoint4[5178] = {X 345.5195, Y 20.4838, Z -5.5000, A 0.000, B 0.000, C 0.000 }
gfCNCPoint4[5179] = {X 344.8326, Y 21.7167, Z -5.5000, A 0.000, B 0.000, C 0.000 }
gfCNCPoint4[5180] = {X 344.0065, Y 22.8611, Z -5.5000, A 0.000, B 0.000, C 0.000 }
gfCNCPoint4[5181] = {X 342.1459, Y 21.3451, Z -5.5000, A 0.000, B 0.000, C 0.000 }
gfCNCPoint4[5182] = {X 341.6015, Y 21.9583, Z -5.5000, A 0.000, B 0.000, C 0.000 }
gfCNCPoint4[5183] = {X 341.0072, Y 22.5232, Z -5.5000, A 0.000, B 0.000, C 0.000 }
gfCNCPoint4[5184] = {X 340.7216, Y 22.7630, Z -5.5000, A 0.000, B 0.000, C 0.000 }
gfCNCPoint4[5185] = {X 340.4270, Y 22.9916, Z -5.5000, A 0.000, B 0.000, C 0.000 }
gfCNCPoint4[5186] = {X 339.6615, Y 23.5549, Z -5.5000, A 0.000, B 0.000, C 0.000 }
gfCNCPoint4[5187] = {X 339.1299, Y 23.9121, Z -5.5000, A 0.000, B 0.000, C 0.000 }
gfCNCPoint4[5188] = {X 338.5759, Y 24.2333, Z -5.5000, A 0.000, B 0.000, C 0.000 }
gfCNCPoint4[5189] = {X 339.6078, Y 24.9035, Z -5.5000, A 0.000, B 0.000, C 0.000 }
gfCNCPoint4[5190] = {X 340.5464, Y 25.6990, Z -5.5000, A 0.000, B 0.000, C 0.000 }
gfCNCPoint4[5191] = {X 341.1849, Y 26.3148, Z -5.5000, A 0.000, B 0.000, C 0.000 }
gfCNCPoint4[5192] = {X 342.1200, Y 27.3788, Z -5.5000, A 0.000, B 0.000, C 0.000 }
gfCNCPoint4[5193] = {X 342.8898, Y 28.5679, Z -5.5000, A 0.000, B 0.000, C 0.000 }
gfCNCPoint4[5194] = {X 343.4778, Y 29.8567, Z -5.5000, A 0.000, B 0.000, C 0.000 }
gfCNCPoint4[5195] = {X 343.8714, Y 31.2174, Z -5.5000, A 0.000, B 0.000, C 0.000 }
gfCNCPoint4[5196] = {X 344.6369, Y 31.6203, Z -5.5000, A 0.000, B 0.000, C 0.000 }
gfCNCPoint4[5197] = {X 345.4580, Y 31.8923, Z -5.5000, A 0.000, B 0.000, C 0.000 }
gfCNCPoint4[5198] = {X 346.3126, Y 32.0261, Z -5.5000, A 0.000, B 0.000, C 0.000 }
gfCNCPoint4[5199] = {X 347.1776, Y 32.0180, Z -5.5000, A 0.000, B 0.000, C 0.000 }
gfCNCPoint4[5200] = {X 347.9597, Y 31.9032, Z -5.5000, A 0.000, B 0.000, C 0.000 }
gfCNCPoint4[5201] = {X 348.6966, Y 31.6174, Z -5.5000, A 0.000, B 0.000, C 0.000 }
gfCNCPoint4[5202] = {X 349.3517, Y 31.1751, Z -5.5000, A 0.000, B 0.000, C 0.000 }
gfCNCPoint4[5203] = {X 350.1527, Y 30.3715, Z -5.5000, A 0.000, B 0.000, C 0.000 }
gfCNCPoint4[5204] = {X 350.8135, Y 29.4491, Z -5.5000, A 0.000, B 0.000, C 0.000 }
gfCNCPoint4[5205] = {X 351.3166, Y 28.4321, Z -5.5000, A 0.000, B 0.000, C 0.000 }
gfCNCPoint4[5206] = {X 351.6489, Y 27.3472, Z -5.5000, A 0.000, B 0.000, C 0.000 }
gfCNCPoint4[5207] = {X 351.8774, Y 25.7621, Z -5.5000, A 0.000, B 0.000, C 0.000 }
gfCNCPoint4[5208] = {X 351.9027, Y 24.1607, Z -5.5000, A 0.000, B 0.000, C 0.000 }
gfCNCPoint4[5209] = {X 351.7244, Y 22.5692, Z -5.5000, A 0.000, B 0.000, C 0.000 }
gfCNCPoint4[5210] = {X 351.4423, Y 21.4555, Z -5.5000, A 0.000, B 0.000, C 0.000 }
gfCNCPoint4[5211] = {X 350.9679, Y 20.4092, Z -5.5000, A 0.000, B 0.000, C 0.000 }
gfCNCPoint4[5212] = {X 350.3161, Y 19.4631, Z -5.5000, A 0.000, B 0.000, C 0.000 }
gfCNCPoint4[5213] = {X 349.6858, Y 18.8475, Z -5.5000, A 0.000, B 0.000, C 0.000 }
gfCNCPoint4[5214] = {X 348.9304, Y 18.3941, Z -5.5000, A 0.000, B 0.000, C 0.000 }
gfCNCPoint4[5215] = {X 348.0907, Y 18.1274, Z -5.5000, A 0.000, B 0.000, C 0.000 }
gfCNCPoint4[5216] = {X 346.9977, Y 17.9944, Z -5.5000, A 0.000, B 0.000, C 0.000 }
gfCNCPoint4[5217] = {X 345.8968, Y 18.0123, Z -5.5000, A 0.000, B 0.000, C 0.000 }
gfCNCPoint4[5218] = {X 344.8086, Y 18.1808, Z -5.5000, A 0.000, B 0.000, C 0.000 }
gfCNCPoint4[5219] = {X 343.7538, Y 18.4967, Z -5.5000, A 0.000, B 0.000, C 0.000 }
gfCNCPoint4[5220] = {X 343.3267, Y 19.5049, Z -5.5000, A 0.000, B 0.000, C 0.000 }
gfCNCPoint4[5221] = {X 342.7884, Y 20.4585, Z -5.5000, A 0.000, B 0.000, C 0.000 }
gfCNCPoint4[5222] = {X 342.1459, Y 21.3451, Z -5.5000, A 0.000, B 0.000, C 0.000 }
gfCNCPoint4[5223] = {X 340.2853, Y 19.8292, Z -5.5000, A 0.000, B 0.000, C 0.000 }
gfCNCPoint4[5224] = {X 339.6794, Y 20.4860, Z -5.5000, A 0.000, B 0.000, C 0.000 }
gfCNCPoint4[5225] = {X 338.9976, Y 21.0636, Z -5.5000, A 0.000, B 0.000, C 0.000 }
gfCNCPoint4[5226] = {X 338.2497, Y 21.6140, Z -5.5000, A 0.000, B 0.000, C 0.000 }
gfCNCPoint4[5227] = {X 337.8538, Y 21.8795, Z -5.5000, A 0.000, B 0.000, C 0.000 }
gfCNCPoint4[5228] = {X 337.4413, Y 22.1185, Z -5.5000, A 0.000, B 0.000, C 0.000 }
gfCNCPoint4[5229] = {X 336.3239, Y 22.6023, Z -5.5000, A 0.000, B 0.000, C 0.000 }
gfCNCPoint4[5230] = {X 335.1415, Y 22.8932, Z -5.5000, A 0.000, B 0.000, C 0.000 }
gfCNCPoint4[5231] = {X 333.9271, Y 22.9829, Z -5.5000, A 0.000, B 0.000, C 0.000 }
gfCNCPoint4[5232] = {X 332.7148, Y 22.8690, Z -5.5000, A 0.000, B 0.000, C 0.000 }
gfCNCPoint4[5233] = {X 331.5384, Y 22.5546, Z -5.5000, A 0.000, B 0.000, C 0.000 }
gfCNCPoint4[5234] = {X 330.4309, Y 22.0485, Z -5.5000, A 0.000, B 0.000, C 0.000 }
gfCNCPoint4[5235] = {X 329.5143, Y 21.4374, Z -5.5000, A 0.000, B 0.000, C 0.000 }
gfCNCPoint4[5236] = {X 328.7005, Y 20.6949, Z -5.5000, A 0.000, B 0.000, C 0.000 }
gfCNCPoint4[5237] = {X 328.0080, Y 19.8382, Z -5.5000, A 0.000, B 0.000, C 0.000 }
gfCNCPoint4[5238] = {X 327.4527, Y 18.8868, Z -5.5000, A 0.000, B 0.000, C 0.000 }
gfCNCPoint4[5239] = {X 323.9321, Y 11.6443, Z -5.5000, A 0.000, B 0.000, C 0.000 }
gfCNCPoint4[5240] = {X 323.5337, Y 10.6421, Z -5.5000, A 0.000, B 0.000, C 0.000 }
gfCNCPoint4[5241] = {X 323.2878, Y 9.5921, Z -5.5000, A 0.000, B 0.000, C 0.000 }
gfCNCPoint4[5242] = {X 323.1997, Y 8.5173, Z -5.5000, A 0.000, B 0.000, C 0.000 }
gfCNCPoint4[5243] = {X 323.2713, Y 7.4413, Z -5.5000, A 0.000, B 0.000, C 0.000 }
gfCNCPoint4[5244] = {X 323.4720, Y 6.4884, Z -5.5000, A 0.000, B 0.000, C 0.000 }
gfCNCPoint4[5245] = {X 323.7980, Y 5.5708, Z -5.5000, A 0.000, B 0.000, C 0.000 }
gfCNCPoint4[5246] = {X 324.2436, Y 4.7049, Z -5.5000, A 0.000, B 0.000, C 0.000 }
gfCNCPoint4[5247] = {X 168.0206, Y 4.7049, Z -5.5000, A 0.000, B 0.000, C 0.000 }
gfCNCPoint4[5248] = {X 168.0206, Y 9.5049, Z -5.5000, A 0.000, B 0.000, C 0.000 }
gfCNCPoint4[5249] = {X 166.5360, Y 9.5049, Z -5.5000, A 0.000, B 0.000, C 0.000 }
gfCNCPoint4[5250] = {X 166.5855, Y 9.9931, Z -5.5000, A 0.000, B 0.000, C 0.000 }
gfCNCPoint4[5251] = {X 166.6021, Y 10.4835, Z -5.5000, A 0.000, B 0.000, C 0.000 }
gfCNCPoint4[5252] = {X 166.6021, Y 13.0969, Z -5.5000, A 0.000, B 0.000, C 0.000 }
gfCNCPoint4[5253] = {X 166.8569, Y 11.8210, Z -5.5000, A 0.000, B 0.000, C 0.000 }
gfCNCPoint4[5254] = {X 167.3349, Y 10.6107, Z -5.5000, A 0.000, B 0.000, C 0.000 }
gfCNCPoint4[5255] = {X 168.0206, Y 9.5049, Z -5.5000, A 0.000, B 0.000, C 0.000 }
gfCNCPoint4[5256] = {X 168.0206, Y 7.1049, Z -5.5000, A 0.000, B 0.000, C 0.000 }
gfCNCPoint4[5257] = {X 162.8434, Y 7.1049, Z -5.5000, A 0.000, B 0.000, C 0.000 }
gfCNCPoint4[5258] = {X 163.4702, Y 7.9131, Z -5.5000, A 0.000, B 0.000, C 0.000 }
gfCNCPoint4[5259] = {X 163.9149, Y 8.8341, Z -5.5000, A 0.000, B 0.000, C 0.000 }
gfCNCPoint4[5260] = {X 164.1578, Y 9.8275, Z -5.5000, A 0.000, B 0.000, C 0.000 }
gfCNCPoint4[5261] = {X 164.1910, Y 10.1548, Z -5.5000, A 0.000, B 0.000, C 0.000 }
gfCNCPoint4[5262] = {X 164.2021, Y 10.4835, Z -5.5000, A 0.000, B 0.000, C 0.000 }
gfCNCPoint4[5263] = {X 164.2021, Y 17.4615, Z -5.5000, A 0.000, B 0.000, C 0.000 }
gfCNCPoint4[5264] = {X 164.1140, Y 18.3847, Z -5.5000, A 0.000, B 0.000, C 0.000 }
gfCNCPoint4[5265] = {X 163.8528, Y 19.2745, Z -5.5000, A 0.000, B 0.000, C 0.000 }
gfCNCPoint4[5266] = {X 163.4281, Y 20.0989, Z -5.5000, A 0.000, B 0.000, C 0.000 }
gfCNCPoint4[5267] = {X 162.8550, Y 20.8280, Z -5.5000, A 0.000, B 0.000, C 0.000 }
gfCNCPoint4[5268] = {X 162.1544, Y 21.4355, Z -5.5000, A 0.000, B 0.000, C 0.000 }
gfCNCPoint4[5269] = {X 161.3515, Y 21.8995, Z -5.5000, A 0.000, B 0.000, C 0.000 }
gfCNCPoint4[5270] = {X 160.4753, Y 22.2033, Z -5.5000, A 0.000, B 0.000, C 0.000 }
gfCNCPoint4[5271] = {X 162.1768, Y 29.1994, Z -5.5000, A 0.000, B 0.000, C 0.000 }
gfCNCPoint4[5272] = {X 161.1137, Y 29.4079, Z -5.5000, A 0.000, B 0.000, C 0.000 }
gfCNCPoint4[5273] = {X 160.0361, Y 29.5204, Z -5.5000, A 0.000, B 0.000, C 0.000 }
gfCNCPoint4[5274] = {X 160.0356, Y 38.3364, Z -5.5000, A 0.000, B 0.000, C 0.000 }
gfCNCPoint4[5275] = {X 160.6838, Y 39.6936, Z -5.5000, A 0.000, B 0.000, C 0.000 }
gfCNCPoint4[5276] = {X 161.1587, Y 41.1206, Z -5.5000, A 0.000, B 0.000, C 0.000 }
gfCNCPoint4[5277] = {X 162.0528, Y 41.1205, Z -5.5000, A 0.000, B 0.000, C 0.000 }
gfCNCPoint4[5278] = {X 161.8705, Y 40.3466, Z -5.5000, A 0.000, B 0.000, C 0.000 }
gfCNCPoint4[5279] = {X 161.7179, Y 39.5663, Z -5.5000, A 0.000, B 0.000, C 0.000 }
gfCNCPoint4[5280] = {X 161.5947, Y 38.7927, Z -5.5000, A 0.000, B 0.000, C 0.000 }
gfCNCPoint4[5281] = {X 161.3802, Y 36.8682, Z -5.5000, A 0.000, B 0.000, C 0.000 }
gfCNCPoint4[5282] = {X 161.3314, Y 34.9324, Z -5.5000, A 0.000, B 0.000, C 0.000 }
gfCNCPoint4[5283] = {X 161.4487, Y 32.9995, Z -5.5000, A 0.000, B 0.000, C 0.000 }
gfCNCPoint4[5284] = {X 161.7312, Y 31.0838, Z -5.5000, A 0.000, B 0.000, C 0.000 }
gfCNCPoint4[5285] = {X 162.1768, Y 29.1994, Z -5.5000, A 0.000, B 0.000, C 0.000 }
gfCNCPoint4[5286] = {X 161.6097, Y 26.8674, Z -5.5000, A 0.000, B 0.000, C 0.000 }
gfCNCPoint4[5287] = {X 160.4740, Y 27.0728, Z -5.5000, A 0.000, B 0.000, C 0.000 }
gfCNCPoint4[5288] = {X 159.3220, Y 27.1415, Z -5.5000, A 0.000, B 0.000, C 0.000 }
gfCNCPoint4[5289] = {X 158.6582, Y 27.1415, Z -5.5000, A 0.000, B 0.000, C 0.000 }
gfCNCPoint4[5290] = {X 158.1465, Y 27.1260, Z -5.5000, A 0.000, B 0.000, C 0.000 }
gfCNCPoint4[5291] = {X 157.6363, Y 27.0835, Z -5.5000, A 0.000, B 0.000, C 0.000 }
gfCNCPoint4[5292] = {X 157.6356, Y 38.9959, Z -5.5000, A 0.000, B 0.000, C 0.000 }
gfCNCPoint4[5293] = {X 158.2194, Y 40.0483, Z -5.5000, A 0.000, B 0.000, C 0.000 }
gfCNCPoint4[5294] = {X 158.6686, Y 41.1648, Z -5.5000, A 0.000, B 0.000, C 0.000 }
gfCNCPoint4[5295] = {X 158.9763, Y 42.3283, Z -5.5000, A 0.000, B 0.000, C 0.000 }
gfCNCPoint4[5296] = {X 159.1376, Y 43.5209, Z -5.5000, A 0.000, B 0.000, C 0.000 }
gfCNCPoint4[5297] = {X 165.4266, Y 43.5200, Z -5.5000, A 0.000, B 0.000, C 0.000 }
gfCNCPoint4[5298] = {X 164.8375, Y 42.0455, Z -5.5000, A 0.000, B 0.000, C 0.000 }
gfCNCPoint4[5299] = {X 164.3779, Y 40.5256, Z -5.5000, A 0.000, B 0.000, C 0.000 }
gfCNCPoint4[5300] = {X 164.2185, Y 39.8499, Z -5.5000, A 0.000, B 0.000, C 0.000 }
gfCNCPoint4[5301] = {X 164.0848, Y 39.1687, Z -5.5000, A 0.000, B 0.000, C 0.000 }
gfCNCPoint4[5302] = {X 163.9656, Y 38.4204, Z -5.5000, A 0.000, B 0.000, C 0.000 }
gfCNCPoint4[5303] = {X 163.7497, Y 36.2695, Z -5.5000, A 0.000, B 0.000, C 0.000 }
gfCNCPoint4[5304] = {X 163.7651, Y 34.1078, Z -5.5000, A 0.000, B 0.000, C 0.000 }
gfCNCPoint4[5305] = {X 164.0116, Y 31.9602, Z -5.5000, A 0.000, B 0.000, C 0.000 }
gfCNCPoint4[5306] = {X 164.4866, Y 29.8513, Z -5.5000, A 0.000, B 0.000, C 0.000 }
gfCNCPoint4[5307] = {X 164.8368, Y 28.7353, Z -5.5000, A 0.000, B 0.000, C 0.000 }
gfCNCPoint4[5308] = {X 165.2511, Y 27.6414, Z -5.5000, A 0.000, B 0.000, C 0.000 }
gfCNCPoint4[5309] = {X 165.8681, Y 26.3087, Z -5.5000, A 0.000, B 0.000, C 0.000 }
gfCNCPoint4[5310] = {X 166.6031, Y 25.0372, Z -5.5000, A 0.000, B 0.000, C 0.000 }
gfCNCPoint4[5311] = {X 167.4500, Y 23.8374, Z -5.5000, A 0.000, B 0.000, C 0.000 }
gfCNCPoint4[5312] = {X 167.1640, Y 23.1367, Z -5.5000, A 0.000, B 0.000, C 0.000 }
gfCNCPoint4[5313] = {X 166.2876, Y 24.1835, Z -5.5000, A 0.000, B 0.000, C 0.000 }
gfCNCPoint4[5314] = {X 165.2726, Y 25.0966, Z -5.5000, A 0.000, B 0.000, C 0.000 }
gfCNCPoint4[5315] = {X 164.1393, Y 25.8578, Z -5.5000, A 0.000, B 0.000, C 0.000 }
gfCNCPoint4[5316] = {X 162.9102, Y 26.4520, Z -5.5000, A 0.000, B 0.000, C 0.000 }
gfCNCPoint4[5317] = {X 161.6097, Y 26.8674, Z -5.5000, A 0.000, B 0.000, C 0.000 }
gfCNCPoint4[5318] = {X 161.0425, Y 24.5353, Z -5.5000, A 0.000, B 0.000, C 0.000 }
gfCNCPoint4[5319] = {X 160.1884, Y 24.6898, Z -5.5000, A 0.000, B 0.000, C 0.000 }
gfCNCPoint4[5320] = {X 159.3220, Y 24.7415, Z -5.5000, A 0.000, B 0.000, C 0.000 }
gfCNCPoint4[5321] = {X 158.6676, Y 24.7415, Z -5.5000, A 0.000, B 0.000, C 0.000 }
gfCNCPoint4[5322] = {X 158.2823, Y 24.7298, Z -5.5000, A 0.000, B 0.000, C 0.000 }
gfCNCPoint4[5323] = {X 157.8982, Y 24.6979, Z -5.5000, A 0.000, B 0.000, C 0.000 }
gfCNCPoint4[5324] = {X 156.9781, Y 24.5368, Z -5.5000, A 0.000, B 0.000, C 0.000 }
gfCNCPoint4[5325] = {X 156.0860, Y 24.2598, Z -5.5000, A 0.000, B 0.000, C 0.000 }
gfCNCPoint4[5326] = {X 155.2365, Y 23.8713, Z -5.5000, A 0.000, B 0.000, C 0.000 }
gfCNCPoint4[5327] = {X 155.2355, Y 39.7518, Z -5.5000, A 0.000, B 0.000, C 0.000 }
gfCNCPoint4[5328] = {X 155.8262, Y 40.6435, Z -5.5000, A 0.000, B 0.000, C 0.000 }
gfCNCPoint4[5329] = {X 156.2805, Y 41.6120, Z -5.5000, A 0.000, B 0.000, C 0.000 }
gfCNCPoint4[5330] = {X 156.5886, Y 42.6363, Z -5.5000, A 0.000, B 0.000, C 0.000 }
gfCNCPoint4[5331] = {X 156.7439, Y 43.6947, Z -5.5000, A 0.000, B 0.000, C 0.000 }
gfCNCPoint4[5332] = {X 156.7579, Y 43.9479, Z -5.5000, A 0.000, B 0.000, C 0.000 }
gfCNCPoint4[5333] = {X 156.7631, Y 44.2015, Z -5.5000, A 0.000, B 0.000, C 0.000 }
gfCNCPoint4[5334] = {X 156.7629, Y 45.0588, Z -5.5000, A 0.000, B 0.000, C 0.000 }
gfCNCPoint4[5335] = {X 156.7352, Y 45.6370, Z -5.5000, A 0.000, B 0.000, C 0.000 }
gfCNCPoint4[5336] = {X 156.6616, Y 46.2112, Z -5.5000, A 0.000, B 0.000, C 0.000 }
gfCNCPoint4[5337] = {X 157.9053, Y 46.0005, Z -5.5000, A 0.000, B 0.000, C 0.000 }
gfCNCPoint4[5338] = {X 159.1642, Y 45.9207, Z -5.5000, A 0.000, B 0.000, C 0.000 }
gfCNCPoint4[5339] = {X 159.2311, Y 45.9202, Z -5.5000, A 0.000, B 0.000, C 0.000 }
gfCNCPoint4[5340] = {X 159.2980, Y 45.9200, Z -5.5000, A 0.000, B 0.000, C 0.000 }
gfCNCPoint4[5341] = {X 169.6795, Y 45.9200, Z -5.5000, A 0.000, B 0.000, C 0.000 }
gfCNCPoint4[5342] = {X 168.8984, Y 44.8498, Z -5.5000, A 0.000, B 0.000, C 0.000 }
gfCNCPoint4[5343] = {X 168.2086, Y 43.7187, Z -5.5000, A 0.000, B 0.000, C 0.000 }
gfCNCPoint4[5344] = {X 167.6148, Y 42.5342, Z -5.5000, A 0.000, B 0.000, C 0.000 }
gfCNCPoint4[5345] = {X 167.1240, Y 41.3128, Z -5.5000, A 0.000, B 0.000, C 0.000 }
gfCNCPoint4[5346] = {X 166.7353, Y 40.0551, Z -5.5000, A 0.000, B 0.000, C 0.000 }
gfCNCPoint4[5347] = {X 166.4515, Y 38.7697, Z -5.5000, A 0.000, B 0.000, C 0.000 }
gfCNCPoint4[5348] = {X 166.3366, Y 38.0483, Z -5.5000, A 0.000, B 0.000, C 0.000 }
gfCNCPoint4[5349] = {X 166.1455, Y 36.1223, Z -5.5000, A 0.000, B 0.000, C 0.000 }
gfCNCPoint4[5350] = {X 166.1648, Y 34.1870, Z -5.5000, A 0.000, B 0.000, C 0.000 }
gfCNCPoint4[5351] = {X 166.3945, Y 32.2652, Z -5.5000, A 0.000, B 0.000, C 0.000 }
gfCNCPoint4[5352] = {X 166.8317, Y 30.3798, Z -5.5000, A 0.000, B 0.000, C 0.000 }
gfCNCPoint4[5353] = {X 167.4713, Y 28.5531, Z -5.5000, A 0.000, B 0.000, C 0.000 }
gfCNCPoint4[5354] = {X 168.2321, Y 26.9827, Z -5.5000, A 0.000, B 0.000, C 0.000 }
gfCNCPoint4[5355] = {X 169.1848, Y 25.5208, Z -5.5000, A 0.000, B 0.000, C 0.000 }
gfCNCPoint4[5356] = {X 170.3141, Y 24.1906, Z -5.5000, A 0.000, B 0.000, C 0.000 }
gfCNCPoint4[5357] = {X 169.9864, Y 23.6221, Z -5.5000, A 0.000, B 0.000, C 0.000 }
gfCNCPoint4[5358] = {X 169.7113, Y 23.0264, Z -5.5000, A 0.000, B 0.000, C 0.000 }
gfCNCPoint4[5359] = {X 167.1001, Y 16.6309, Z -5.5000, A 0.000, B 0.000, C 0.000 }
gfCNCPoint4[5360] = {X 166.7820, Y 15.6636, Z -5.5000, A 0.000, B 0.000, C 0.000 }
gfCNCPoint4[5361] = {X 166.6021, Y 14.6613, Z -5.5000, A 0.000, B 0.000, C 0.000 }
gfCNCPoint4[5362] = {X 166.6021, Y 17.4615, Z -5.5000, A 0.000, B 0.000, C 0.000 }
gfCNCPoint4[5363] = {X 166.5130, Y 18.5970, Z -5.5000, A 0.000, B 0.000, C 0.000 }
gfCNCPoint4[5364] = {X 166.2479, Y 19.7047, Z -5.5000, A 0.000, B 0.000, C 0.000 }
gfCNCPoint4[5365] = {X 165.8132, Y 20.7575, Z -5.5000, A 0.000, B 0.000, C 0.000 }
gfCNCPoint4[5366] = {X 165.2197, Y 21.7296, Z -5.5000, A 0.000, B 0.000, C 0.000 }
gfCNCPoint4[5367] = {X 164.3790, Y 22.6986, Z -5.5000, A 0.000, B 0.000, C 0.000 }
gfCNCPoint4[5368] = {X 163.3812, Y 23.5049, Z -5.5000, A 0.000, B 0.000, C 0.000 }
gfCNCPoint4[5369] = {X 162.2574, Y 24.1235, Z -5.5000, A 0.000, B 0.000, C 0.000 }
gfCNCPoint4[5370] = {X 161.0425, Y 24.5353, Z -5.5000, A 0.000, B 0.000, C 0.000 }
gfCNCPoint4[5371] = {X 160.4753, Y 22.2033, Z -5.5000, A 0.000, B 0.000, C 0.000 }
gfCNCPoint4[5372] = {X 159.9028, Y 22.3069, Z -5.5000, A 0.000, B 0.000, C 0.000 }
gfCNCPoint4[5373] = {X 159.3220, Y 22.3415, Z -5.5000, A 0.000, B 0.000, C 0.000 }
gfCNCPoint4[5374] = {X 158.6770, Y 22.3415, Z -5.5000, A 0.000, B 0.000, C 0.000 }
gfCNCPoint4[5375] = {X 157.8802, Y 22.2733, Z -5.5000, A 0.000, B 0.000, C 0.000 }
gfCNCPoint4[5376] = {X 157.1050, Y 22.0767, Z -5.5000, A 0.000, B 0.000, C 0.000 }
gfCNCPoint4[5377] = {X 156.3719, Y 21.7569, Z -5.5000, A 0.000, B 0.000, C 0.000 }
gfCNCPoint4[5378] = {X 155.5229, Y 21.1791, Z -5.5000, A 0.000, B 0.000, C 0.000 }
gfCNCPoint4[5379] = {X 154.8125, Y 20.4374, Z -5.5000, A 0.000, B 0.000, C 0.000 }
gfCNCPoint4[5380] = {X 152.8367, Y 20.4381, Z -5.5000, A 0.000, B 0.000, C 0.000 }
gfCNCPoint4[5381] = {X 152.8355, Y 40.6542, Z -5.5000, A 0.000, B 0.000, C 0.000 }
gfCNCPoint4[5382] = {X 153.1750, Y 41.0214, Z -5.5000, A 0.000, B 0.000, C 0.000 }
gfCNCPoint4[5383] = {X 153.6799, Y 41.7255, Z -5.5000, A 0.000, B 0.000, C 0.000 }
gfCNCPoint4[5384] = {X 154.0533, Y 42.5075, Z -5.5000, A 0.000, B 0.000, C 0.000 }
gfCNCPoint4[5385] = {X 154.2834, Y 43.3428, Z -5.5000, A 0.000, B 0.000, C 0.000 }
gfCNCPoint4[5386] = {X 154.3631, Y 44.2057, Z -5.5000, A 0.000, B 0.000, C 0.000 }
gfCNCPoint4[5387] = {X 154.3629, Y 45.0469, Z -5.5000, A 0.000, B 0.000, C 0.000 }
gfCNCPoint4[5388] = {X 154.3440, Y 45.4307, Z -5.5000, A 0.000, B 0.000, C 0.000 }
gfCNCPoint4[5389] = {X 154.2951, Y 45.8119, Z -5.5000, A 0.000, B 0.000, C 0.000 }
gfCNCPoint4[5390] = {X 154.0370, Y 46.7541, Z -5.5000, A 0.000, B 0.000, C 0.000 }
gfCNCPoint4[5391] = {X 153.5963, Y 47.6260, Z -5.5000, A 0.000, B 0.000, C 0.000 }
gfCNCPoint4[5392] = {X 152.9909, Y 48.3926, Z -5.5000, A 0.000, B 0.000, C 0.000 }
gfCNCPoint4[5393] = {X 152.2448, Y 49.0233, Z -5.5000, A 0.000, B 0.000, C 0.000 }
gfCNCPoint4[5394] = {X 151.3881, Y 49.4928, Z -5.5000, A 0.000, B 0.000, C 0.000 }
gfCNCPoint4[5395] = {X 150.4551, Y 49.7822, Z -5.5000, A 0.000, B 0.000, C 0.000 }
gfCNCPoint4[5396] = {X 149.4831, Y 49.8800, Z -5.5000, A 0.000, B 0.000, C 0.000 }
gfCNCPoint4[5397] = {X 143.0396, Y 49.8800, Z -5.5000, A 0.000, B 0.000, C 0.000 }
gfCNCPoint4[5398] = {X 142.0923, Y 49.7872, Z -5.5000, A 0.000, B 0.000, C 0.000 }
gfCNCPoint4[5399] = {X 141.1811, Y 49.5122, Z -5.5000, A 0.000, B 0.000, C 0.000 }
gfCNCPoint4[5400] = {X 140.3405, Y 49.0656, Z -5.5000, A 0.000, B 0.000, C 0.000 }
gfCNCPoint4[5401] = {X 139.6026, Y 48.4643, Z -5.5000, A 0.000, B 0.000, C 0.000 }
gfCNCPoint4[5402] = {X 138.9955, Y 47.7312, Z -5.5000, A 0.000, B 0.000, C 0.000 }
gfCNCPoint4[5403] = {X 138.5423, Y 46.8942, Z -5.5000, A 0.000, B 0.000, C 0.000 }
gfCNCPoint4[5404] = {X 138.2601, Y 45.9852, Z -5.5000, A 0.000, B 0.000, C 0.000 }
gfCNCPoint4[5405] = {X 138.1598, Y 45.0386, Z -5.5000, A 0.000, B 0.000, C 0.000 }
gfCNCPoint4[5406] = {X 138.1601, Y 44.1417, Z -5.5000, A 0.000, B 0.000, C 0.000 }
gfCNCPoint4[5407] = {X 138.2148, Y 43.4769, Z -5.5000, A 0.000, B 0.000, C 0.000 }
gfCNCPoint4[5408] = {X 138.3597, Y 42.8258, Z -5.5000, A 0.000, B 0.000, C 0.000 }
gfCNCPoint4[5409] = {X 129.1532, Y 40.1052, Z -5.5000, A 0.000, B 0.000, C 0.000 }
gfCNCPoint4[5410] = {X 129.5665, Y 38.9035, Z -5.5000, A 0.000, B 0.000, C 0.000 }
gfCNCPoint4[5411] = {X 130.0836, Y 37.7426, Z -5.5000, A 0.000, B 0.000, C 0.000 }
gfCNCPoint4[5412] = {X 130.0836, Y 31.6021, Z -5.5000, A 0.000, B 0.000, C 0.000 }
gfCNCPoint4[5413] = {X 129.2063, Y 31.3797, Z -5.5000, A 0.000, B 0.000, C 0.000 }
gfCNCPoint4[5414] = {X 128.3447, Y 31.1030, Z -5.5000, A 0.000, B 0.000, C 0.000 }
gfCNCPoint4[5415] = {X 128.3444, Y 38.3297, Z -5.5000, A 0.000, B 0.000, C 0.000 }
gfCNCPoint4[5416] = {X 128.7847, Y 39.2011, Z -5.5000, A 0.000, B 0.000, C 0.000 }
gfCNCPoint4[5417] = {X 129.1532, Y 40.1052, Z -5.5000, A 0.000, B 0.000, C 0.000 }
gfCNCPoint4[5418] = {X 131.4548, Y 40.7854, Z -5.5000, A 0.000, B 0.000, C 0.000 }
gfCNCPoint4[5419] = {X 131.9017, Y 39.5320, Z -5.5000, A 0.000, B 0.000, C 0.000 }
gfCNCPoint4[5420] = {X 132.4836, Y 38.3354, Z -5.5000, A 0.000, B 0.000, C 0.000 }
gfCNCPoint4[5421] = {X 132.4836, Y 29.5202, Z -5.5000, A 0.000, B 0.000, C 0.000 }
gfCNCPoint4[5422] = {X 131.3526, Y 29.3993, Z -5.5000, A 0.000, B 0.000, C 0.000 }
gfCNCPoint4[5423] = {X 130.2379, Y 29.1726, Z -5.5000, A 0.000, B 0.000, C 0.000 }
gfCNCPoint4[5424] = {X 129.1495, Y 28.8420, Z -5.5000, A 0.000, B 0.000, C 0.000 }
gfCNCPoint4[5425] = {X 128.0251, Y 28.3767, Z -5.5000, A 0.000, B 0.000, C 0.000 }
gfCNCPoint4[5426] = {X 126.9533, Y 27.8006, Z -5.5000, A 0.000, B 0.000, C 0.000 }
gfCNCPoint4[5427] = {X 125.9448, Y 27.1196, Z -5.5000, A 0.000, B 0.000, C 0.000 }
gfCNCPoint4[5428] = {X 125.9444, Y 38.9902, Z -5.5000, A 0.000, B 0.000, C 0.000 }
gfCNCPoint4[5429] = {X 126.4740, Y 39.9288, Z -5.5000, A 0.000, B 0.000, C 0.000 }
gfCNCPoint4[5430] = {X 126.8960, Y 40.9205, Z -5.5000, A 0.000, B 0.000, C 0.000 }
gfCNCPoint4[5431] = {X 127.2098, Y 41.9730, Z -5.5000, A 0.000, B 0.000, C 0.000 }
gfCNCPoint4[5432] = {X 127.4025, Y 43.0542, Z -5.5000, A 0.000, B 0.000, C 0.000 }
gfCNCPoint4[5433] = {X 127.4714, Y 44.1502, Z -5.5000, A 0.000, B 0.000, C 0.000 }
gfCNCPoint4[5434] = {X 127.4716, Y 45.0000, Z -5.5000, A 0.000, B 0.000, C 0.000 }
gfCNCPoint4[5435] = {X 127.4070, Y 46.1159, Z -5.5000, A 0.000, B 0.000, C 0.000 }
gfCNCPoint4[5436] = {X 127.2143, Y 47.2168, Z -5.5000, A 0.000, B 0.000, C 0.000 }
gfCNCPoint4[5437] = {X 126.8960, Y 48.2883, Z -5.5000, A 0.000, B 0.000, C 0.000 }
gfCNCPoint4[5438] = {X 126.2883, Y 49.6376, Z -5.5000, A 0.000, B 0.000, C 0.000 }
gfCNCPoint4[5439] = {X 125.4821, Y 50.8786, Z -5.5000, A 0.000, B 0.000, C 0.000 }
gfCNCPoint4[5440] = {X 124.4962, Y 51.9821, Z -5.5000, A 0.000, B 0.000, C 0.000 }
gfCNCPoint4[5441] = {X 123.3536, Y 52.9225, Z -5.5000, A 0.000, B 0.000, C 0.000 }
gfCNCPoint4[5442] = {X 122.0810, Y 53.6778, Z -5.5000, A 0.000, B 0.000, C 0.000 }
gfCNCPoint4[5443] = {X 120.7081, Y 54.2302, Z -5.5000, A 0.000, B 0.000, C 0.000 }
gfCNCPoint4[5444] = {X 119.2671, Y 54.5669, Z -5.5000, A 0.000, B 0.000, C 0.000 }
gfCNCPoint4[5445] = {X 117.7916, Y 54.6800, Z -5.5000, A 0.000, B 0.000, C 0.000 }
gfCNCPoint4[5446] = {X 111.9185, Y 54.6800, Z -5.5000, A 0.000, B 0.000, C 0.000 }
gfCNCPoint4[5447] = {X 111.7445, Y 54.6784, Z -5.5000, A 0.000, B 0.000, C 0.000 }
gfCNCPoint4[5448] = {X 111.5706, Y 54.6737, Z -5.5000, A 0.000, B 0.000, C 0.000 }
gfCNCPoint4[5449] = {X 111.0530, Y 69.0644, Z -5.5000, A 0.000, B 0.000, C 0.000 }
gfCNCPoint4[5450] = {X 109.0268, Y 68.9057, Z -5.5000, A 0.000, B 0.000, C 0.000 }
gfCNCPoint4[5451] = {X 107.0213, Y 68.5768, Z -5.5000, A 0.000, B 0.000, C 0.000 }
gfCNCPoint4[5452] = {X 105.0765, Y 68.8983, Z -5.5000, A 0.000, B 0.000, C 0.000 }
gfCNCPoint4[5453] = {X 103.1119, Y 69.0597, Z -5.5000, A 0.000, B 0.000, C 0.000 }
gfCNCPoint4[5454] = {X 101.1407, Y 69.0599, Z -5.5000, A 0.000, B 0.000, C 0.000 }
gfCNCPoint4[5455] = {X 99.1761, Y 68.8989, Z -5.5000, A 0.000, B 0.000, C 0.000 }
gfCNCPoint4[5456] = {X 97.2313, Y 68.5777, Z -5.5000, A 0.000, B 0.000, C 0.000 }
gfCNCPoint4[5457] = {X 95.6131, Y 68.8563, Z -5.5000, A 0.000, B 0.000, C 0.000 }
gfCNCPoint4[5458] = {X 93.9796, Y 69.0240, Z -5.5000, A 0.000, B 0.000, C 0.000 }
gfCNCPoint4[5459] = {X 92.3385, Y 69.0800, Z -5.5000, A 0.000, B 0.000, C 0.000 }
gfCNCPoint4[5460] = {X 86.6884, Y 69.0800, Z -5.5000, A 0.000, B 0.000, C 0.000 }
gfCNCPoint4[5461] = {X 84.7316, Y 70.2669, Z -5.5000, A 0.000, B 0.000, C 0.000 }
gfCNCPoint4[5462] = {X 82.6870, Y 71.2951, Z -5.5000, A 0.000, B 0.000, C 0.000 }
gfCNCPoint4[5463] = {X 107.2677, Y 71.2951, Z -5.5000, A 0.000, B 0.000, C 0.000 }
gfCNCPoint4[5464] = {X 109.1211, Y 70.1132, Z -5.5000, A 0.000, B 0.000, C 0.000 }
gfCNCPoint4[5465] = {X 111.0530, Y 69.0644, Z -5.5000, A 0.000, B 0.000, C 0.000 }
gfCNCPoint4[5466] = {X 111.1392, Y 66.6660, Z -5.5000, A 0.000, B 0.000, C 0.000 }
gfCNCPoint4[5467] = {X 109.0671, Y 66.4917, Z -5.5000, A 0.000, B 0.000, C 0.000 }
gfCNCPoint4[5468] = {X 107.0213, Y 66.1197, Z -5.5000, A 0.000, B 0.000, C 0.000 }
gfCNCPoint4[5469] = {X 105.0796, Y 66.4776, Z -5.5000, A 0.000, B 0.000, C 0.000 }
gfCNCPoint4[5470] = {X 103.1135, Y 66.6574, Z -5.5000, A 0.000, B 0.000, C 0.000 }
gfCNCPoint4[5471] = {X 101.1392, Y 66.6576, Z -5.5000, A 0.000, B 0.000, C 0.000 }
gfCNCPoint4[5472] = {X 99.1730, Y 66.4782, Z -5.5000, A 0.000, B 0.000, C 0.000 }
gfCNCPoint4[5473] = {X 97.2313, Y 66.1207, Z -5.5000, A 0.000, B 0.000, C 0.000 }
gfCNCPoint4[5474] = {X 95.6161, Y 66.4308, Z -5.5000, A 0.000, B 0.000, C 0.000 }
gfCNCPoint4[5475] = {X 93.9821, Y 66.6176, Z -5.5000, A 0.000, B 0.000, C 0.000 }
gfCNCPoint4[5476] = {X 92.3385, Y 66.6800, Z -5.5000, A 0.000, B 0.000, C 0.000 }
gfCNCPoint4[5477] = {X 85.9487, Y 66.6800, Z -5.5000, A 0.000, B 0.000, C 0.000 }
gfCNCPoint4[5478] = {X 83.8779, Y 67.9935, Z -5.5000, A 0.000, B 0.000, C 0.000 }
gfCNCPoint4[5479] = {X 81.6945, Y 69.1099, Z -5.5000, A 0.000, B 0.000, C 0.000 }
gfCNCPoint4[5480] = {X 79.6015, Y 69.9548, Z -5.5000, A 0.000, B 0.000, C 0.000 }
gfCNCPoint4[5481] = {X 77.4442, Y 70.6184, Z -5.5000, A 0.000, B 0.000, C 0.000 }
gfCNCPoint4[5482] = {X 75.2382, Y 71.0959, Z -5.5000, A 0.000, B 0.000, C 0.000 }
gfCNCPoint4[5483] = {X 72.9995, Y 71.3838, Z -5.5000, A 0.000, B 0.000, C 0.000 }
gfCNCPoint4[5484] = {X 70.7445, Y 71.4800, Z -5.5000, A 0.000, B 0.000, C 0.000 }
gfCNCPoint4[5485] = {X 64.1851, Y 71.4800, Z -5.5000, A 0.000, B 0.000, C 0.000 }
gfCNCPoint4[5486] = {X 62.0752, Y 71.3958, Z -5.5000, A 0.000, B 0.000, C 0.000 }
gfCNCPoint4[5487] = {X 59.9787, Y 71.1438, Z -5.5000, A 0.000, B 0.000, C 0.000 }
gfCNCPoint4[5488] = {X 57.9089, Y 70.7255, Z -5.5000, A 0.000, B 0.000, C 0.000 }
gfCNCPoint4[5489] = {X 55.8790, Y 70.1436, Z -5.5000, A 0.000, B 0.000, C 0.000 }
gfCNCPoint4[5490] = {X 53.8492, Y 70.7255, Z -5.5000, A 0.000, B 0.000, C 0.000 }
gfCNCPoint4[5491] = {X 51.7794, Y 71.1438, Z -5.5000, A 0.000, B 0.000, C 0.000 }
gfCNCPoint4[5492] = {X 49.6829, Y 71.3958, Z -5.5000, A 0.000, B 0.000, C 0.000 }
gfCNCPoint4[5493] = {X 47.5729, Y 71.4800, Z -5.5000, A 0.000, B 0.000, C 0.000 }
gfCNCPoint4[5494] = {X 40.6393, Y 71.4800, Z -5.5000, A 0.000, B 0.000, C 0.000 }
gfCNCPoint4[5495] = {X 38.8053, Y 71.4164, Z -5.5000, A 0.000, B 0.000, C 0.000 }
gfCNCPoint4[5496] = {X 36.9802, Y 71.2260, Z -5.5000, A 0.000, B 0.000, C 0.000 }
gfCNCPoint4[5497] = {X 34.3996, Y 72.0352, Z -5.5000, A 0.000, B 0.000, C 0.000 }
gfCNCPoint4[5498] = {X 31.7580, Y 72.6151, Z -5.5000, A 0.000, B 0.000, C 0.000 }
gfCNCPoint4[5499] = {X 30.3326, Y 73.1748, Z -5.5000, A 0.000, B 0.000, C 0.000 }
gfCNCPoint4[5500] = {X 28.8923, Y 73.6951, Z -5.5000, A 0.000, B 0.000, C 0.000 }
gfCNCPoint4[5501] = {X 108.0302, Y 73.6951, Z -5.5000, A 0.000, B 0.000, C 0.000 }
gfCNCPoint4[5502] = {X 110.0252, Y 72.3689, Z -5.5000, A 0.000, B 0.000, C 0.000 }
gfCNCPoint4[5503] = {X 112.1232, Y 71.2126, Z -5.5000, A 0.000, B 0.000, C 0.000 }
gfCNCPoint4[5504] = {X 113.1260, Y 70.7368, Z -5.5000, A 0.000, B 0.000, C 0.000 }
gfCNCPoint4[5505] = {X 114.1463, Y 70.2999, Z -5.5000, A 0.000, B 0.000, C 0.000 }
gfCNCPoint4[5506] = {X 117.4427, Y 66.6800, Z -5.5000, A 0.000, B 0.000, C 0.000 }
gfCNCPoint4[5507] = {X 111.9185, Y 66.6800, Z -5.5000, A 0.000, B 0.000, C 0.000 }
gfCNCPoint4[5508] = {X 111.5288, Y 66.6765, Z -5.5000, A 0.000, B 0.000, C 0.000 }
gfCNCPoint4[5509] = {X 111.1392, Y 66.6660, Z -5.5000, A 0.000, B 0.000, C 0.000 }
gfCNCPoint4[5510] = {X 111.2255, Y 64.2675, Z -5.5000, A 0.000, B 0.000, C 0.000 }
gfCNCPoint4[5511] = {X 109.1063, Y 64.0738, Z -5.5000, A 0.000, B 0.000, C 0.000 }
gfCNCPoint4[5512] = {X 107.0213, Y 63.6477, Z -5.5000, A 0.000, B 0.000, C 0.000 }
gfCNCPoint4[5513] = {X 105.0841, Y 64.0514, Z -5.5000, A 0.000, B 0.000, C 0.000 }
gfCNCPoint4[5514] = {X 103.1158, Y 64.2545, Z -5.5000, A 0.000, B 0.000, C 0.000 }
gfCNCPoint4[5515] = {X 101.1370, Y 64.2547, Z -5.5000, A 0.000, B 0.000, C 0.000 }
gfCNCPoint4[5516] = {X 99.1686, Y 64.0521, Z -5.5000, A 0.000, B 0.000, C 0.000 }
gfCNCPoint4[5517] = {X 97.2313, Y 63.6488, Z -5.5000, A 0.000, B 0.000, C 0.000 }
gfCNCPoint4[5518] = {X 95.6204, Y 63.9986, Z -5.5000, A 0.000, B 0.000, C 0.000 }
gfCNCPoint4[5519] = {X 93.9855, Y 64.2095, Z -5.5000, A 0.000, B 0.000, C 0.000 }
gfCNCPoint4[5520] = {X 92.3385, Y 64.2800, Z -5.5000, A 0.000, B 0.000, C 0.000 }
gfCNCPoint4[5521] = {X 85.8951, Y 64.2800, Z -5.5000, A 0.000, B 0.000, C 0.000 }
gfCNCPoint4[5522] = {X 85.5417, Y 64.2768, Z -5.5000, A 0.000, B 0.000, C 0.000 }
gfCNCPoint4[5523] = {X 85.1884, Y 64.2670, Z -5.5000, A 0.000, B 0.000, C 0.000 }
gfCNCPoint4[5524] = {X 83.3593, Y 65.5113, Z -5.5000, A 0.000, B 0.000, C 0.000 }
gfCNCPoint4[5525] = {X 81.4238, Y 66.5824, Z -5.5000, A 0.000, B 0.000, C 0.000 }
gfCNCPoint4[5526] = {X 79.3981, Y 67.4713, Z -5.5000, A 0.000, B 0.000, C 0.000 }
gfCNCPoint4[5527] = {X 77.2994, Y 68.1706, Z -5.5000, A 0.000, B 0.000, C 0.000 }
gfCNCPoint4[5528] = {X 75.1454, Y 68.6744, Z -5.5000, A 0.000, B 0.000, C 0.000 }
gfCNCPoint4[5529] = {X 72.9543, Y 68.9784, Z -5.5000, A 0.000, B 0.000, C 0.000 }
gfCNCPoint4[5530] = {X 70.7445, Y 69.0800, Z -5.5000, A 0.000, B 0.000, C 0.000 }
gfCNCPoint4[5531] = {X 64.1851, Y 69.0800, Z -5.5000, A 0.000, B 0.000, C 0.000 }
gfCNCPoint4[5532] = {X 62.0678, Y 68.9867, Z -5.5000, A 0.000, B 0.000, C 0.000 }
gfCNCPoint4[5533] = {X 59.9669, Y 68.7076, Z -5.5000, A 0.000, B 0.000, C 0.000 }
gfCNCPoint4[5534] = {X 57.8986, Y 68.2449, Z -5.5000, A 0.000, B 0.000, C 0.000 }
gfCNCPoint4[5535] = {X 55.8790, Y 67.6021, Z -5.5000, A 0.000, B 0.000, C 0.000 }
gfCNCPoint4[5536] = {X 53.8595, Y 68.2449, Z -5.5000, A 0.000, B 0.000, C 0.000 }
gfCNCPoint4[5537] = {X 51.7912, Y 68.7076, Z -5.5000, A 0.000, B 0.000, C 0.000 }
gfCNCPoint4[5538] = {X 49.6903, Y 68.9867, Z -5.5000, A 0.000, B 0.000, C 0.000 }
gfCNCPoint4[5539] = {X 47.5729, Y 69.0800, Z -5.5000, A 0.000, B 0.000, C 0.000 }
gfCNCPoint4[5540] = {X 40.6393, Y 69.0800, Z -5.5000, A 0.000, B 0.000, C 0.000 }
gfCNCPoint4[5541] = {X 38.6748, Y 68.9997, Z -5.5000, A 0.000, B 0.000, C 0.000 }
gfCNCPoint4[5542] = {X 36.7235, Y 68.7595, Z -5.5000, A 0.000, B 0.000, C 0.000 }
gfCNCPoint4[5543] = {X 34.8831, Y 69.3993, Z -5.5000, A 0.000, B 0.000, C 0.000 }
gfCNCPoint4[5544] = {X 33.0033, Y 69.9114, Z -5.5000, A 0.000, B 0.000, C 0.000 }
gfCNCPoint4[5545] = {X 31.0928, Y 70.2936, Z -5.5000, A 0.000, B 0.000, C 0.000 }
gfCNCPoint4[5546] = {X 29.6089, Y 70.8826, Z -5.5000, A 0.000, B 0.000, C 0.000 }
gfCNCPoint4[5547] = {X 28.1080, Y 71.4268, Z -5.5000, A 0.000, B 0.000, C 0.000 }
gfCNCPoint4[5548] = {X 27.6115, Y 71.5958, Z -5.5000, A 0.000, B 0.000, C 0.000 }
gfCNCPoint4[5549] = {X 27.1133, Y 71.7598, Z -5.5000, A 0.000, B 0.000, C 0.000 }
gfCNCPoint4[5550] = {X 25.5166, Y 72.2528, Z -5.5000, A 0.000, B 0.000, C 0.000 }
gfCNCPoint4[5551] = {X 23.9034, Y 72.6885, Z -5.5000, A 0.000, B 0.000, C 0.000 }
gfCNCPoint4[5552] = {X 23.9034, Y 76.0951, Z -5.5000, A 0.000, B 0.000, C 0.000 }
gfCNCPoint4[5553] = {X 108.8286, Y 76.0951, Z -5.5000, A 0.000, B 0.000, C 0.000 }
gfCNCPoint4[5554] = {X 110.4001, Y 74.9718, Z -5.5000, A 0.000, B 0.000, C 0.000 }
gfCNCPoint4[5555] = {X 112.0493, Y 73.9662, Z -5.5000, A 0.000, B 0.000, C 0.000 }
gfCNCPoint4[5556] = {X 113.7674, Y 73.0834, Z -5.5000, A 0.000, B 0.000, C 0.000 }
gfCNCPoint4[5557] = {X 115.5453, Y 72.3282, Z -5.5000, A 0.000, B 0.000, C 0.000 }
gfCNCPoint4[5558] = {X 123.7269, Y 63.3437, Z -5.5000, A 0.000, B 0.000, C 0.000 }
gfCNCPoint4[5559] = {X 121.7847, Y 63.8620, Z -5.5000, A 0.000, B 0.000, C 0.000 }
gfCNCPoint4[5560] = {X 119.7990, Y 64.1752, Z -5.5000, A 0.000, B 0.000, C 0.000 }
gfCNCPoint4[5561] = {X 117.7916, Y 64.2800, Z -5.5000, A 0.000, B 0.000, C 0.000 }
gfCNCPoint4[5562] = {X 111.9185, Y 64.2800, Z -5.5000, A 0.000, B 0.000, C 0.000 }
gfCNCPoint4[5563] = {X 111.5719, Y 64.2769, Z -5.5000, A 0.000, B 0.000, C 0.000 }
gfCNCPoint4[5564] = {X 111.2255, Y 64.2675, Z -5.5000, A 0.000, B 0.000, C 0.000 }
gfCNCPoint4[5565] = {X 111.3118, Y 61.8691, Z -5.5000, A 0.000, B 0.000, C 0.000 }
gfCNCPoint4[5566] = {X 109.8628, Y 61.7544, Z -5.5000, A 0.000, B 0.000, C 0.000 }
gfCNCPoint4[5567] = {X 108.4291, Y 61.5154, Z -5.5000, A 0.000, B 0.000, C 0.000 }
gfCNCPoint4[5568] = {X 107.0213, Y 61.1540, Z -5.5000, A 0.000, B 0.000, C 0.000 }
gfCNCPoint4[5569] = {X 105.0907, Y 61.6173, Z -5.5000, A 0.000, B 0.000, C 0.000 }
gfCNCPoint4[5570] = {X 103.1191, Y 61.8506, Z -5.5000, A 0.000, B 0.000, C 0.000 }
gfCNCPoint4[5571] = {X 101.1337, Y 61.8509, Z -5.5000, A 0.000, B 0.000, C 0.000 }
gfCNCPoint4[5572] = {X 99.1620, Y 61.6181, Z -5.5000, A 0.000, B 0.000, C 0.000 }
gfCNCPoint4[5573] = {X 97.2313, Y 61.1553, Z -5.5000, A 0.000, B 0.000, C 0.000 }
gfCNCPoint4[5574] = {X 95.6267, Y 61.5566, Z -5.5000, A 0.000, B 0.000, C 0.000 }
gfCNCPoint4[5575] = {X 93.9906, Y 61.7990, Z -5.5000, A 0.000, B 0.000, C 0.000 }
gfCNCPoint4[5576] = {X 92.3385, Y 61.8800, Z -5.5000, A 0.000, B 0.000, C 0.000 }
gfCNCPoint4[5577] = {X 85.8951, Y 61.8800, Z -5.5000, A 0.000, B 0.000, C 0.000 }
gfCNCPoint4[5578] = {X 85.1609, Y 61.8640, Z -5.5000, A 0.000, B 0.000, C 0.000 }
gfCNCPoint4[5579] = {X 84.4280, Y 61.8161, Z -5.5000, A 0.000, B 0.000, C 0.000 }
gfCNCPoint4[5580] = {X 82.7247, Y 63.0692, Z -5.5000, A 0.000, B 0.000, C 0.000 }
gfCNCPoint4[5581] = {X 80.9073, Y 64.1504, Z -5.5000, A 0.000, B 0.000, C 0.000 }
gfCNCPoint4[5582] = {X 78.9932, Y 65.0494, Z -5.5000, A 0.000, B 0.000, C 0.000 }
gfCNCPoint4[5583] = {X 77.0007, Y 65.7577, Z -5.5000, A 0.000, B 0.000, C 0.000 }
gfCNCPoint4[5584] = {X 74.9487, Y 66.2685, Z -5.5000, A 0.000, B 0.000, C 0.000 }
gfCNCPoint4[5585] = {X 72.8566, Y 66.5769, Z -5.5000, A 0.000, B 0.000, C 0.000 }
gfCNCPoint4[5586] = {X 70.7445, Y 66.6800, Z -5.5000, A 0.000, B 0.000, C 0.000 }
gfCNCPoint4[5587] = {X 64.1851, Y 66.6800, Z -5.5000, A 0.000, B 0.000, C 0.000 }
gfCNCPoint4[5588] = {X 62.0576, Y 66.5754, Z -5.5000, A 0.000, B 0.000, C 0.000 }
gfCNCPoint4[5589] = {X 59.9505, Y 66.2624, Z -5.5000, A 0.000, B 0.000, C 0.000 }
gfCNCPoint4[5590] = {X 57.8844, Y 65.7442, Z -5.5000, A 0.000, B 0.000, C 0.000 }
gfCNCPoint4[5591] = {X 55.8790, Y 65.0258, Z -5.5000, A 0.000, B 0.000, C 0.000 }
gfCNCPoint4[5592] = {X 53.8737, Y 65.7442, Z -5.5000, A 0.000, B 0.000, C 0.000 }
gfCNCPoint4[5593] = {X 51.8075, Y 66.2624, Z -5.5000, A 0.000, B 0.000, C 0.000 }
gfCNCPoint4[5594] = {X 49.7005, Y 66.5753, Z -5.5000, A 0.000, B 0.000, C 0.000 }
gfCNCPoint4[5595] = {X 47.5729, Y 66.6800, Z -5.5000, A 0.000, B 0.000, C 0.000 }
gfCNCPoint4[5596] = {X 40.6393, Y 66.6800, Z -5.5000, A 0.000, B 0.000, C 0.000 }
gfCNCPoint4[5597] = {X 38.5449, Y 66.5786, Z -5.5000, A 0.000, B 0.000, C 0.000 }
gfCNCPoint4[5598] = {X 36.4701, Y 66.2753, Z -5.5000, A 0.000, B 0.000, C 0.000 }
gfCNCPoint4[5599] = {X 34.5052, Y 67.0014, Z -5.5000, A 0.000, B 0.000, C 0.000 }
gfCNCPoint4[5600] = {X 32.4883, Y 67.5670, Z -5.5000, A 0.000, B 0.000, C 0.000 }
gfCNCPoint4[5601] = {X 30.4324, Y 67.9685, Z -5.5000, A 0.000, B 0.000, C 0.000 }
gfCNCPoint4[5602] = {X 28.4168, Y 68.7666, Z -5.5000, A 0.000, B 0.000, C 0.000 }
gfCNCPoint4[5603] = {X 26.3692, Y 69.4781, Z -5.5000, A 0.000, B 0.000, C 0.000 }
gfCNCPoint4[5604] = {X 23.9547, Y 70.1962, Z -5.5000, A 0.000, B 0.000, C 0.000 }
gfCNCPoint4[5605] = {X 21.5034, Y 70.7763, Z -5.5000, A 0.000, B 0.000, C 0.000 }
gfCNCPoint4[5606] = {X 21.5034, Y 78.4951, Z -5.5000, A 0.000, B 0.000, C 0.000 }
gfCNCPoint4[5607] = {X 109.6685, Y 78.4951, Z -5.5000, A 0.000, B 0.000, C 0.000 }
gfCNCPoint4[5608] = {X 111.3412, Y 77.2320, Z -5.5000, A 0.000, B 0.000, C 0.000 }
gfCNCPoint4[5609] = {X 113.1174, Y 76.1191, Z -5.5000, A 0.000, B 0.000, C 0.000 }
gfCNCPoint4[5610] = {X 114.9837, Y 75.1650, Z -5.5000, A 0.000, B 0.000, C 0.000 }
gfCNCPoint4[5611] = {X 116.9258, Y 74.3767, Z -5.5000, A 0.000, B 0.000, C 0.000 }
gfCNCPoint4[5612] = {X 130.4109, Y 59.5682, Z -5.5000, A 0.000, B 0.000, C 0.000 }
gfCNCPoint4[5613] = {X 129.5277, Y 58.7530, Z -5.5000, A 0.000, B 0.000, C 0.000 }
gfCNCPoint4[5614] = {X 128.6970, Y 57.8844, Z -5.5000, A 0.000, B 0.000, C 0.000 }
gfCNCPoint4[5615] = {X 127.3928, Y 58.8835, Z -5.5000, A 0.000, B 0.000, C 0.000 }
gfCNCPoint4[5616] = {X 125.9976, Y 59.7511, Z -5.5000, A 0.000, B 0.000, C 0.000 }
gfCNCPoint4[5617] = {X 124.5247, Y 60.4790, Z -5.5000, A 0.000, B 0.000, C 0.000 }
gfCNCPoint4[5618] = {X 122.9880, Y 61.0602, Z -5.5000, A 0.000, B 0.000, C 0.000 }
gfCNCPoint4[5619] = {X 121.2876, Y 61.5140, Z -5.5000, A 0.000, B 0.000, C 0.000 }
gfCNCPoint4[5620] = {X 119.5491, Y 61.7883, Z -5.5000, A 0.000, B 0.000, C 0.000 }
gfCNCPoint4[5621] = {X 117.7916, Y 61.8800, Z -5.5000, A 0.000, B 0.000, C 0.000 }
gfCNCPoint4[5622] = {X 111.9185, Y 61.8800, Z -5.5000, A 0.000, B 0.000, C 0.000 }
gfCNCPoint4[5623] = {X 111.6151, Y 61.8773, Z -5.5000, A 0.000, B 0.000, C 0.000 }
gfCNCPoint4[5624] = {X 111.3118, Y 61.8691, Z -5.5000, A 0.000, B 0.000, C 0.000 }
gfCNCPoint4[5625] = {X 111.3980, Y 59.4706, Z -5.5000, A 0.000, B 0.000, C 0.000 }
gfCNCPoint4[5626] = {X 109.9127, Y 59.3404, Z -5.5000, A 0.000, B 0.000, C 0.000 }
gfCNCPoint4[5627] = {X 108.4486, Y 59.0581, Z -5.5000, A 0.000, B 0.000, C 0.000 }
gfCNCPoint4[5628] = {X 107.0213, Y 58.6267, Z -5.5000, A 0.000, B 0.000, C 0.000 }
gfCNCPoint4[5629] = {X 105.4260, Y 59.0985, Z -5.5000, A 0.000, B 0.000, C 0.000 }
gfCNCPoint4[5630] = {X 103.7872, Y 59.3842, Z -5.5000, A 0.000, B 0.000, C 0.000 }
gfCNCPoint4[5631] = {X 102.1264, Y 59.4800, Z -5.5000, A 0.000, B 0.000, C 0.000 }
gfCNCPoint4[5632] = {X 100.4656, Y 59.3847, Z -5.5000, A 0.000, B 0.000, C 0.000 }
gfCNCPoint4[5633] = {X 98.8267, Y 59.0996, Z -5.5000, A 0.000, B 0.000, C 0.000 }
gfCNCPoint4[5634] = {X 97.2313, Y 58.6283, Z -5.5000, A 0.000, B 0.000, C 0.000 }
gfCNCPoint4[5635] = {X 95.6367, Y 59.0994, Z -5.5000, A 0.000, B 0.000, C 0.000 }
gfCNCPoint4[5636] = {X 93.9986, Y 59.3845, Z -5.5000, A 0.000, B 0.000, C 0.000 }
gfCNCPoint4[5637] = {X 92.3385, Y 59.4800, Z -5.5000, A 0.000, B 0.000, C 0.000 }
gfCNCPoint4[5638] = {X 85.8951, Y 59.4800, Z -5.5000, A 0.000, B 0.000, C 0.000 }
gfCNCPoint4[5639] = {X 84.7780, Y 59.4368, Z -5.5000, A 0.000, B 0.000, C 0.000 }
gfCNCPoint4[5640] = {X 83.6677, Y 59.3077, Z -5.5000, A 0.000, B 0.000, C 0.000 }
gfCNCPoint4[5641] = {X 82.0978, Y 60.5827, Z -5.5000, A 0.000, B 0.000, C 0.000 }
gfCNCPoint4[5642] = {X 80.4031, Y 61.6862, Z -5.5000, A 0.000, B 0.000, C 0.000 }
gfCNCPoint4[5643] = {X 78.6021, Y 62.6061, Z -5.5000, A 0.000, B 0.000, C 0.000 }
gfCNCPoint4[5644] = {X 76.7146, Y 63.3324, Z -5.5000, A 0.000, B 0.000, C 0.000 }
gfCNCPoint4[5645] = {X 74.7614, Y 63.8569, Z -5.5000, A 0.000, B 0.000, C 0.000 }
gfCNCPoint4[5646] = {X 72.7641, Y 64.1739, Z -5.5000, A 0.000, B 0.000, C 0.000 }
gfCNCPoint4[5647] = {X 70.7445, Y 64.2800, Z -5.5000, A 0.000, B 0.000, C 0.000 }
gfCNCPoint4[5648] = {X 64.1851, Y 64.2800, Z -5.5000, A 0.000, B 0.000, C 0.000 }
gfCNCPoint4[5649] = {X 62.0428, Y 64.1606, Z -5.5000, A 0.000, B 0.000, C 0.000 }
gfCNCPoint4[5650] = {X 59.9269, Y 63.8039, Z -5.5000, A 0.000, B 0.000, C 0.000 }
gfCNCPoint4[5651] = {X 57.8638, Y 63.2143, Z -5.5000, A 0.000, B 0.000, C 0.000 }
gfCNCPoint4[5652] = {X 55.8790, Y 62.3991, Z -5.5000, A 0.000, B 0.000, C 0.000 }
gfCNCPoint4[5653] = {X 53.8942, Y 63.2143, Z -5.5000, A 0.000, B 0.000, C 0.000 }
gfCNCPoint4[5654] = {X 51.8311, Y 63.8039, Z -5.5000, A 0.000, B 0.000, C 0.000 }
gfCNCPoint4[5655] = {X 49.7153, Y 64.1606, Z -5.5000, A 0.000, B 0.000, C 0.000 }
gfCNCPoint4[5656] = {X 47.5729, Y 64.2800, Z -5.5000, A 0.000, B 0.000, C 0.000 }
gfCNCPoint4[5657] = {X 40.6393, Y 64.2800, Z -5.5000, A 0.000, B 0.000, C 0.000 }
gfCNCPoint4[5658] = {X 39.1550, Y 64.2228, Z -5.5000, A 0.000, B 0.000, C 0.000 }
gfCNCPoint4[5659] = {X 37.6795, Y 64.0514, Z -5.5000, A 0.000, B 0.000, C 0.000 }
gfCNCPoint4[5660] = {X 36.2215, Y 63.7670, Z -5.5000, A 0.000, B 0.000, C 0.000 }
gfCNCPoint4[5661] = {X 34.1362, Y 64.5946, Z -5.5000, A 0.000, B 0.000, C 0.000 }
gfCNCPoint4[5662] = {X 31.9818, Y 65.2205, Z -5.5000, A 0.000, B 0.000, C 0.000 }
gfCNCPoint4[5663] = {X 29.7778, Y 65.6391, Z -5.5000, A 0.000, B 0.000, C 0.000 }
gfCNCPoint4[5664] = {X 27.7192, Y 66.4653, Z -5.5000, A 0.000, B 0.000, C 0.000 }
gfCNCPoint4[5665] = {X 25.6250, Y 67.1964, Z -5.5000, A 0.000, B 0.000, C 0.000 }
gfCNCPoint4[5666] = {X 23.4802, Y 67.8385, Z -5.5000, A 0.000, B 0.000, C 0.000 }
gfCNCPoint4[5667] = {X 21.3043, Y 68.3656, Z -5.5000, A 0.000, B 0.000, C 0.000 }
gfCNCPoint4[5668] = {X 19.1034, Y 68.7761, Z -5.5000, A 0.000, B 0.000, C 0.000 }
gfCNCPoint4[5669] = {X 19.1034, Y 80.8951, Z -5.5000, A 0.000, B 0.000, C 0.000 }
gfCNCPoint4[5670] = {X 110.5571, Y 80.8951, Z -5.5000, A 0.000, B 0.000, C 0.000 }
gfCNCPoint4[5671] = {X 112.3055, Y 79.4886, Z -5.5000, A 0.000, B 0.000, C 0.000 }
gfCNCPoint4[5672] = {X 114.1900, Y 78.2704, Z -5.5000, A 0.000, B 0.000, C 0.000 }
gfCNCPoint4[5673] = {X 116.1903, Y 77.2535, Z -5.5000, A 0.000, B 0.000, C 0.000 }
gfCNCPoint4[5674] = {X 118.2849, Y 76.4488, Z -5.5000, A 0.000, B 0.000, C 0.000 }
gfCNCPoint4[5675] = {X 133.9631, Y 59.2320, Z -5.5000, A 0.000, B 0.000, C 0.000 }
gfCNCPoint4[5676] = {X 132.7153, Y 58.3545, Z -5.5000, A 0.000, B 0.000, C 0.000 }
gfCNCPoint4[5677] = {X 131.5520, Y 57.3680, Z -5.5000, A 0.000, B 0.000, C 0.000 }
gfCNCPoint4[5678] = {X 130.4824, Y 56.2805, Z -5.5000, A 0.000, B 0.000, C 0.000 }
gfCNCPoint4[5679] = {X 129.6655, Y 55.2988, Z -5.5000, A 0.000, B 0.000, C 0.000 }
gfCNCPoint4[5680] = {X 128.9251, Y 54.2582, Z -5.5000, A 0.000, B 0.000, C 0.000 }
gfCNCPoint4[5681] = {X 128.0750, Y 55.1942, Z -5.5000, A 0.000, B 0.000, C 0.000 }
gfCNCPoint4[5682] = {X 127.1464, Y 56.0525, Z -5.5000, A 0.000, B 0.000, C 0.000 }
gfCNCPoint4[5683] = {X 125.7915, Y 57.0695, Z -5.5000, A 0.000, B 0.000, C 0.000 }
gfCNCPoint4[5684] = {X 124.3270, Y 57.9212, Z -5.5000, A 0.000, B 0.000, C 0.000 }
gfCNCPoint4[5685] = {X 122.7731, Y 58.5961, Z -5.5000, A 0.000, B 0.000, C 0.000 }
gfCNCPoint4[5686] = {X 121.1510, Y 59.0849, Z -5.5000, A 0.000, B 0.000, C 0.000 }
gfCNCPoint4[5687] = {X 119.4828, Y 59.3809, Z -5.5000, A 0.000, B 0.000, C 0.000 }
gfCNCPoint4[5688] = {X 117.7916, Y 59.4800, Z -5.5000, A 0.000, B 0.000, C 0.000 }
gfCNCPoint4[5689] = {X 111.9185, Y 59.4800, Z -5.5000, A 0.000, B 0.000, C 0.000 }
gfCNCPoint4[5690] = {X 111.6582, Y 59.4777, Z -5.5000, A 0.000, B 0.000, C 0.000 }
gfCNCPoint4[5691] = {X 111.3980, Y 59.4706, Z -5.5000, A 0.000, B 0.000, C 0.000 }
gfCNCPoint4[5692] = {X 111.4843, Y 57.0722, Z -5.5000, A 0.000, B 0.000, C 0.000 }
gfCNCPoint4[5693] = {X 109.9569, Y 56.9197, Z -5.5000, A 0.000, B 0.000, C 0.000 }
gfCNCPoint4[5694] = {X 108.4612, Y 56.5747, Z -5.5000, A 0.000, B 0.000, C 0.000 }
gfCNCPoint4[5695] = {X 107.0213, Y 56.0428, Z -5.5000, A 0.000, B 0.000, C 0.000 }
gfCNCPoint4[5696] = {X 105.4432, Y 56.6151, Z -5.5000, A 0.000, B 0.000, C 0.000 }
gfCNCPoint4[5697] = {X 103.8010, Y 56.9630, Z -5.5000, A 0.000, B 0.000, C 0.000 }
gfCNCPoint4[5698] = {X 102.1265, Y 57.0800, Z -5.5000, A 0.000, B 0.000, C 0.000 }
gfCNCPoint4[5699] = {X 100.4519, Y 56.9637, Z -5.5000, A 0.000, B 0.000, C 0.000 }
gfCNCPoint4[5700] = {X 98.8096, Y 56.6164, Z -5.5000, A 0.000, B 0.000, C 0.000 }
gfCNCPoint4[5701] = {X 97.2313, Y 56.0448, Z -5.5000, A 0.000, B 0.000, C 0.000 }
gfCNCPoint4[5702] = {X 95.6538, Y 56.6162, Z -5.5000, A 0.000, B 0.000, C 0.000 }
gfCNCPoint4[5703] = {X 94.0123, Y 56.9635, Z -5.5000, A 0.000, B 0.000, C 0.000 }
gfCNCPoint4[5704] = {X 92.3385, Y 57.0800, Z -5.5000, A 0.000, B 0.000, C 0.000 }
gfCNCPoint4[5705] = {X 85.8951, Y 57.0800, Z -5.5000, A 0.000, B 0.000, C 0.000 }
gfCNCPoint4[5706] = {X 84.3894, Y 56.9858, Z -5.5000, A 0.000, B 0.000, C 0.000 }
gfCNCPoint4[5707] = {X 82.9073, Y 56.7047, Z -5.5000, A 0.000, B 0.000, C 0.000 }
gfCNCPoint4[5708] = {X 81.4846, Y 58.0224, Z -5.5000, A 0.000, B 0.000, C 0.000 }
gfCNCPoint4[5709] = {X 79.9203, Y 59.1682, Z -5.5000, A 0.000, B 0.000, C 0.000 }
gfCNCPoint4[5710] = {X 78.2348, Y 60.1271, Z -5.5000, A 0.000, B 0.000, C 0.000 }
gfCNCPoint4[5711] = {X 76.4504, Y 60.8863, Z -5.5000, A 0.000, B 0.000, C 0.000 }
gfCNCPoint4[5712] = {X 74.5908, Y 61.4359, Z -5.5000, A 0.000, B 0.000, C 0.000 }
gfCNCPoint4[5713] = {X 72.6804, Y 61.7686, Z -5.5000, A 0.000, B 0.000, C 0.000 }
gfCNCPoint4[5714] = {X 70.7445, Y 61.8800, Z -5.5000, A 0.000, B 0.000, C 0.000 }
gfCNCPoint4[5715] = {X 64.1851, Y 61.8800, Z -5.5000, A 0.000, B 0.000, C 0.000 }
gfCNCPoint4[5716] = {X 62.4514, Y 61.7907, Z -5.5000, A 0.000, B 0.000, C 0.000 }
gfCNCPoint4[5717] = {X 60.7359, Y 61.5238, Z -5.5000, A 0.000, B 0.000, C 0.000 }
gfCNCPoint4[5718] = {X 59.0570, Y 61.0822, Z -5.5000, A 0.000, B 0.000, C 0.000 }
gfCNCPoint4[5719] = {X 57.4323, Y 60.4704, Z -5.5000, A 0.000, B 0.000, C 0.000 }
gfCNCPoint4[5720] = {X 55.8790, Y 59.6950, Z -5.5000, A 0.000, B 0.000, C 0.000 }
gfCNCPoint4[5721] = {X 54.3258, Y 60.4704, Z -5.5000, A 0.000, B 0.000, C 0.000 }
gfCNCPoint4[5722] = {X 52.7011, Y 61.0822, Z -5.5000, A 0.000, B 0.000, C 0.000 }
gfCNCPoint4[5723] = {X 51.0221, Y 61.5238, Z -5.5000, A 0.000, B 0.000, C 0.000 }
gfCNCPoint4[5724] = {X 49.3067, Y 61.7907, Z -5.5000, A 0.000, B 0.000, C 0.000 }
gfCNCPoint4[5725] = {X 47.5729, Y 61.8800, Z -5.5000, A 0.000, B 0.000, C 0.000 }
gfCNCPoint4[5726] = {X 40.6393, Y 61.8800, Z -5.5000, A 0.000, B 0.000, C 0.000 }
gfCNCPoint4[5727] = {X 39.0679, Y 61.8067, Z -5.5000, A 0.000, B 0.000, C 0.000 }
gfCNCPoint4[5728] = {X 37.5102, Y 61.5874, Z -5.5000, A 0.000, B 0.000, C 0.000 }
gfCNCPoint4[5729] = {X 35.9796, Y 61.2241, Z -5.5000, A 0.000, B 0.000, C 0.000 }
gfCNCPoint4[5730] = {X 34.3397, Y 61.9604, Z -5.5000, A 0.000, B 0.000, C 0.000 }
gfCNCPoint4[5731] = {X 32.6434, Y 62.5552, Z -5.5000, A 0.000, B 0.000, C 0.000 }
gfCNCPoint4[5732] = {X 30.9028, Y 63.0043, Z -5.5000, A 0.000, B 0.000, C 0.000 }
gfCNCPoint4[5733] = {X 29.1304, Y 63.3043, Z -5.5000, A 0.000, B 0.000, C 0.000 }
gfCNCPoint4[5734] = {X 27.0255, Y 64.1619, Z -5.5000, A 0.000, B 0.000, C 0.000 }
gfCNCPoint4[5735] = {X 24.8808, Y 64.9147, Z -5.5000, A 0.000, B 0.000, C 0.000 }
gfCNCPoint4[5736] = {X 22.1986, Y 65.6930, Z -5.5000, A 0.000, B 0.000, C 0.000 }
gfCNCPoint4[5737] = {X 19.4683, Y 66.2806, Z -5.5000, A 0.000, B 0.000, C 0.000 }
gfCNCPoint4[5738] = {X 16.7034, Y 66.6746, Z -5.5000, A 0.000, B 0.000, C 0.000 }
gfCNCPoint4[5739] = {X 16.7034, Y 83.2951, Z -5.5000, A 0.000, B 0.000, C 0.000 }
gfCNCPoint4[5740] = {X 111.5041, Y 83.2951, Z -5.5000, A 0.000, B 0.000, C 0.000 }
gfCNCPoint4[5741] = {X 112.9236, Y 82.0343, Z -5.5000, A 0.000, B 0.000, C 0.000 }
gfCNCPoint4[5742] = {X 114.4601, Y 80.9193, Z -5.5000, A 0.000, B 0.000, C 0.000 }
gfCNCPoint4[5743] = {X 116.0988, Y 79.9608, Z -5.5000, A 0.000, B 0.000, C 0.000 }
gfCNCPoint4[5744] = {X 117.8239, Y 79.1681, Z -5.5000, A 0.000, B 0.000, C 0.000 }
gfCNCPoint4[5745] = {X 119.6186, Y 78.5489, Z -5.5000, A 0.000, B 0.000, C 0.000 }
gfCNCPoint4[5746] = {X 137.8568, Y 58.5207, Z -5.5000, A 0.000, B 0.000, C 0.000 }
gfCNCPoint4[5747] = {X 136.5221, Y 57.9303, Z -5.5000, A 0.000, B 0.000, C 0.000 }
gfCNCPoint4[5748] = {X 135.2536, Y 57.2085, Z -5.5000, A 0.000, B 0.000, C 0.000 }
gfCNCPoint4[5749] = {X 134.0097, Y 56.3195, Z -5.5000, A 0.000, B 0.000, C 0.000 }
gfCNCPoint4[5750] = {X 132.8665, Y 55.3043, Z -5.5000, A 0.000, B 0.000, C 0.000 }
gfCNCPoint4[5751] = {X 131.8368, Y 54.1742, Z -5.5000, A 0.000, B 0.000, C 0.000 }
gfCNCPoint4[5752] = {X 130.9319, Y 52.9419, Z -5.5000, A 0.000, B 0.000, C 0.000 }
gfCNCPoint4[5753] = {X 130.2147, Y 51.7225, Z -5.5000, A 0.000, B 0.000, C 0.000 }
gfCNCPoint4[5754] = {X 129.6199, Y 50.4390, Z -5.5000, A 0.000, B 0.000, C 0.000 }
gfCNCPoint4[5755] = {X 129.1532, Y 49.1035, Z -5.5000, A 0.000, B 0.000, C 0.000 }
gfCNCPoint4[5756] = {X 128.6036, Y 50.3877, Z -5.5000, A 0.000, B 0.000, C 0.000 }
gfCNCPoint4[5757] = {X 127.9093, Y 51.5998, Z -5.5000, A 0.000, B 0.000, C 0.000 }
gfCNCPoint4[5758] = {X 127.0798, Y 52.7237, Z -5.5000, A 0.000, B 0.000, C 0.000 }
gfCNCPoint4[5759] = {X 126.0417, Y 53.8239, Z -5.5000, A 0.000, B 0.000, C 0.000 }
gfCNCPoint4[5760] = {X 124.8743, Y 54.7858, Z -5.5000, A 0.000, B 0.000, C 0.000 }
gfCNCPoint4[5761] = {X 123.5958, Y 55.5942, Z -5.5000, A 0.000, B 0.000, C 0.000 }
gfCNCPoint4[5762] = {X 122.2263, Y 56.2365, Z -5.5000, A 0.000, B 0.000, C 0.000 }
gfCNCPoint4[5763] = {X 120.7872, Y 56.7027, Z -5.5000, A 0.000, B 0.000, C 0.000 }
gfCNCPoint4[5764] = {X 119.3012, Y 56.9853, Z -5.5000, A 0.000, B 0.000, C 0.000 }
gfCNCPoint4[5765] = {X 117.7916, Y 57.0800, Z -5.5000, A 0.000, B 0.000, C 0.000 }
gfCNCPoint4[5766] = {X 111.9185, Y 57.0800, Z -5.5000, A 0.000, B 0.000, C 0.000 }
gfCNCPoint4[5767] = {X 111.7014, Y 57.0780, Z -5.5000, A 0.000, B 0.000, C 0.000 }
gfCNCPoint4[5768] = {X 111.4843, Y 57.0722, Z -5.5000, A 0.000, B 0.000, C 0.000 }
gfCNCPoint4[5769] = {X 111.5706, Y 54.6737, Z -5.5000, A 0.000, B 0.000, C 0.000 }
gfCNCPoint4[5770] = {X 110.3804, Y 54.5570, Z -5.5000, A 0.000, B 0.000, C 0.000 }
gfCNCPoint4[5771] = {X 109.2137, Y 54.2944, Z -5.5000, A 0.000, B 0.000, C 0.000 }
gfCNCPoint4[5772] = {X 108.0882, Y 53.8900, Z -5.5000, A 0.000, B 0.000, C 0.000 }
gfCNCPoint4[5773] = {X 107.0213, Y 53.3498, Z -5.5000, A 0.000, B 0.000, C 0.000 }
gfCNCPoint4[5774] = {X 106.6480, Y 53.5578, Z -5.5000, A 0.000, B 0.000, C 0.000 }
gfCNCPoint4[5775] = {X 106.2658, Y 53.7492, Z -5.5000, A 0.000, B 0.000, C 0.000 }
gfCNCPoint4[5776] = {X 105.0149, Y 54.2383, Z -5.5000, A 0.000, B 0.000, C 0.000 }
gfCNCPoint4[5777] = {X 103.7084, Y 54.5495, Z -5.5000, A 0.000, B 0.000, C 0.000 }
gfCNCPoint4[5778] = {X 102.3713, Y 54.6768, Z -5.5000, A 0.000, B 0.000, C 0.000 }
gfCNCPoint4[5779] = {X 101.0295, Y 54.6179, Z -5.5000, A 0.000, B 0.000, C 0.000 }
gfCNCPoint4[5780] = {X 99.7088, Y 54.3738, Z -5.5000, A 0.000, B 0.000, C 0.000 }
gfCNCPoint4[5781] = {X 98.4345, Y 53.9493, Z -5.5000, A 0.000, B 0.000, C 0.000 }
gfCNCPoint4[5782] = {X 97.2313, Y 53.3524, Z -5.5000, A 0.000, B 0.000, C 0.000 }
gfCNCPoint4[5783] = {X 96.0852, Y 53.9255, Z -5.5000, A 0.000, B 0.000, C 0.000 }
gfCNCPoint4[5784] = {X 94.8734, Y 54.3422, Z -5.5000, A 0.000, B 0.000, C 0.000 }
gfCNCPoint4[5785] = {X 93.6172, Y 54.5952, Z -5.5000, A 0.000, B 0.000, C 0.000 }
gfCNCPoint4[5786] = {X 92.3385, Y 54.6800, Z -5.5000, A 0.000, B 0.000, C 0.000 }
gfCNCPoint4[5787] = {X 85.8951, Y 54.6800, Z -5.5000, A 0.000, B 0.000, C 0.000 }
gfCNCPoint4[5788] = {X 84.6159, Y 54.5951, Z -5.5000, A 0.000, B 0.000, C 0.000 }
gfCNCPoint4[5789] = {X 83.3592, Y 54.3419, Z -5.5000, A 0.000, B 0.000, C 0.000 }
gfCNCPoint4[5790] = {X 82.1469, Y 53.9249, Z -5.5000, A 0.000, B 0.000, C 0.000 }
gfCNCPoint4[5791] = {X 81.0644, Y 55.1572, Z -5.5000, A 0.000, B 0.000, C 0.000 }
gfCNCPoint4[5792] = {X 79.8495, Y 56.2591, Z -5.5000, A 0.000, B 0.000, C 0.000 }
gfCNCPoint4[5793] = {X 78.5178, Y 57.2166, Z -5.5000, A 0.000, B 0.000, C 0.000 }
gfCNCPoint4[5794] = {X 77.0863, Y 58.0174, Z -5.5000, A 0.000, B 0.000, C 0.000 }
gfCNCPoint4[5795] = {X 75.5734, Y 58.6511, Z -5.5000, A 0.000, B 0.000, C 0.000 }
gfCNCPoint4[5796] = {X 73.9986, Y 59.1096, Z -5.5000, A 0.000, B 0.000, C 0.000 }
gfCNCPoint4[5797] = {X 72.3820, Y 59.3871, Z -5.5000, A 0.000, B 0.000, C 0.000 }
gfCNCPoint4[5798] = {X 70.7445, Y 59.4800, Z -5.5000, A 0.000, B 0.000, C 0.000 }
gfCNCPoint4[5799] = {X 64.1851, Y 59.4800, Z -5.5000, A 0.000, B 0.000, C 0.000 }
gfCNCPoint4[5800] = {X 62.4203, Y 59.3720, Z -5.5000, A 0.000, B 0.000, C 0.000 }
gfCNCPoint4[5801] = {X 60.6818, Y 59.0498, Z -5.5000, A 0.000, B 0.000, C 0.000 }
gfCNCPoint4[5802] = {X 58.9955, Y 58.5181, Z -5.5000, A 0.000, B 0.000, C 0.000 }
gfCNCPoint4[5803] = {X 57.3866, Y 57.7848, Z -5.5000, A 0.000, B 0.000, C 0.000 }
gfCNCPoint4[5804] = {X 55.8790, Y 56.8608, Z -5.5000, A 0.000, B 0.000, C 0.000 }
gfCNCPoint4[5805] = {X 54.3715, Y 57.7848, Z -5.5000, A 0.000, B 0.000, C 0.000 }
gfCNCPoint4[5806] = {X 52.7626, Y 58.5181, Z -5.5000, A 0.000, B 0.000, C 0.000 }
gfCNCPoint4[5807] = {X 51.0763, Y 59.0498, Z -5.5000, A 0.000, B 0.000, C 0.000 }
gfCNCPoint4[5808] = {X 49.3378, Y 59.3720, Z -5.5000, A 0.000, B 0.000, C 0.000 }
gfCNCPoint4[5809] = {X 47.5729, Y 59.4800, Z -5.5000, A 0.000, B 0.000, C 0.000 }
gfCNCPoint4[5810] = {X 40.6393, Y 59.4800, Z -5.5000, A 0.000, B 0.000, C 0.000 }
gfCNCPoint4[5811] = {X 38.9797, Y 59.3846, Z -5.5000, A 0.000, B 0.000, C 0.000 }
gfCNCPoint4[5812] = {X 37.3420, Y 59.0996, Z -5.5000, A 0.000, B 0.000, C 0.000 }
gfCNCPoint4[5813] = {X 35.7478, Y 58.6288, Z -5.5000, A 0.000, B 0.000, C 0.000 }
gfCNCPoint4[5814] = {X 34.0329, Y 59.4874, Z -5.5000, A 0.000, B 0.000, C 0.000 }
gfCNCPoint4[5815] = {X 32.2395, Y 60.1670, Z -5.5000, A 0.000, B 0.000, C 0.000 }
gfCNCPoint4[5816] = {X 30.3862, Y 60.6605, Z -5.5000, A 0.000, B 0.000, C 0.000 }
gfCNCPoint4[5817] = {X 28.4923, Y 60.9627, Z -5.5000, A 0.000, B 0.000, C 0.000 }
gfCNCPoint4[5818] = {X 26.3368, Y 61.8560, Z -5.5000, A 0.000, B 0.000, C 0.000 }
gfCNCPoint4[5819] = {X 24.1366, Y 62.6330, Z -5.5000, A 0.000, B 0.000, C 0.000 }
gfCNCPoint4[5820] = {X 21.7299, Y 63.3359, Z -5.5000, A 0.000, B 0.000, C 0.000 }
gfCNCPoint4[5821] = {X 19.2814, Y 63.8753, Z -5.5000, A 0.000, B 0.000, C 0.000 }
gfCNCPoint4[5822] = {X 16.8022, Y 64.2487, Z -5.5000, A 0.000, B 0.000, C 0.000 }
gfCNCPoint4[5823] = {X 14.3034, Y 64.4545, Z -5.5000, A 0.000, B 0.000, C 0.000 }
gfCNCPoint4[5824] = {X 14.3034, Y 85.6951, Z -5.5000, A 0.000, B 0.000, C 0.000 }
gfCNCPoint4[5825] = {X 112.5228, Y 85.6951, Z -5.5000, A 0.000, B 0.000, C 0.000 }
gfCNCPoint4[5826] = {X 113.9423, Y 84.3098, Z -5.5000, A 0.000, B 0.000, C 0.000 }
gfCNCPoint4[5827] = {X 115.5145, Y 83.1005, Z -5.5000, A 0.000, B 0.000, C 0.000 }
gfCNCPoint4[5828] = {X 117.2177, Y 82.0840, Z -5.5000, A 0.000, B 0.000, C 0.000 }
gfCNCPoint4[5829] = {X 119.0283, Y 81.2744, Z -5.5000, A 0.000, B 0.000, C 0.000 }
gfCNCPoint4[5830] = {X 120.9214, Y 80.6827, Z -5.5000, A 0.000, B 0.000, C 0.000 }
gfCNCPoint4[5831] = {X 142.4288, Y 57.0645, Z -5.5000, A 0.000, B 0.000, C 0.000 }
gfCNCPoint4[5832] = {X 141.1659, Y 56.9338, Z -5.5000, A 0.000, B 0.000, C 0.000 }
gfCNCPoint4[5833] = {X 139.9236, Y 56.6712, Z -5.5000, A 0.000, B 0.000, C 0.000 }
gfCNCPoint4[5834] = {X 138.7158, Y 56.2797, Z -5.5000, A 0.000, B 0.000, C 0.000 }
gfCNCPoint4[5835] = {X 137.2788, Y 55.6179, Z -5.5000, A 0.000, B 0.000, C 0.000 }
gfCNCPoint4[5836] = {X 135.9406, Y 54.7740, Z -5.5000, A 0.000, B 0.000, C 0.000 }
gfCNCPoint4[5837] = {X 134.7242, Y 53.7624, Z -5.5000, A 0.000, B 0.000, C 0.000 }
gfCNCPoint4[5838] = {X 133.6504, Y 52.6006, Z -5.5000, A 0.000, B 0.000, C 0.000 }
gfCNCPoint4[5839] = {X 132.7376, Y 51.3084, Z -5.5000, A 0.000, B 0.000, C 0.000 }
gfCNCPoint4[5840] = {X 132.0016, Y 49.9080, Z -5.5000, A 0.000, B 0.000, C 0.000 }
gfCNCPoint4[5841] = {X 131.4549, Y 48.4234, Z -5.5000, A 0.000, B 0.000, C 0.000 }
gfCNCPoint4[5842] = {X 131.1845, Y 47.3200, Z -5.5000, A 0.000, B 0.000, C 0.000 }
gfCNCPoint4[5843] = {X 131.0190, Y 46.1961, Z -5.5000, A 0.000, B 0.000, C 0.000 }
gfCNCPoint4[5844] = {X 130.9598, Y 45.0616, Z -5.5000, A 0.000, B 0.000, C 0.000 }
gfCNCPoint4[5845] = {X 130.9601, Y 44.0979, Z -5.5000, A 0.000, B 0.000, C 0.000 }
gfCNCPoint4[5846] = {X 131.0921, Y 42.4244, Z -5.5000, A 0.000, B 0.000, C 0.000 }
gfCNCPoint4[5847] = {X 131.4548, Y 40.7854, Z -5.5000, A 0.000, B 0.000, C 0.000 }
gfCNCPoint4[5848] = {X 133.7565, Y 41.4655, Z -5.5000, A 0.000, B 0.000, C 0.000 }
gfCNCPoint4[5849] = {X 134.2330, Y 40.1906, Z -5.5000, A 0.000, B 0.000, C 0.000 }
gfCNCPoint4[5850] = {X 134.8836, Y 38.9952, Z -5.5000, A 0.000, B 0.000, C 0.000 }
gfCNCPoint4[5851] = {X 134.8836, Y 27.0854, Z -5.5000, A 0.000, B 0.000, C 0.000 }
gfCNCPoint4[5852] = {X 134.3931, Y 27.1259, Z -5.5000, A 0.000, B 0.000, C 0.000 }
gfCNCPoint4[5853] = {X 133.9011, Y 27.1414, Z -5.5000, A 0.000, B 0.000, C 0.000 }
gfCNCPoint4[5854] = {X 133.2006, Y 27.1415, Z -5.5000, A 0.000, B 0.000, C 0.000 }
gfCNCPoint4[5855] = {X 131.9567, Y 27.0613, Z -5.5000, A 0.000, B 0.000, C 0.000 }
gfCNCPoint4[5856] = {X 130.7334, Y 26.8218, Z -5.5000, A 0.000, B 0.000, C 0.000 }
gfCNCPoint4[5857] = {X 129.5510, Y 26.4272, Z -5.5000, A 0.000, B 0.000, C 0.000 }
gfCNCPoint4[5858] = {X 128.4291, Y 25.8838, Z -5.5000, A 0.000, B 0.000, C 0.000 }
gfCNCPoint4[5859] = {X 127.3864, Y 25.2008, Z -5.5000, A 0.000, B 0.000, C 0.000 }
gfCNCPoint4[5860] = {X 126.3457, Y 24.2962, Z -5.5000, A 0.000, B 0.000, C 0.000 }
gfCNCPoint4[5861] = {X 125.4442, Y 23.2528, Z -5.5000, A 0.000, B 0.000, C 0.000 }
gfCNCPoint4[5862] = {X 124.7000, Y 22.0920, Z -5.5000, A 0.000, B 0.000, C 0.000 }
gfCNCPoint4[5863] = {X 124.1283, Y 20.8372, Z -5.5000, A 0.000, B 0.000, C 0.000 }
gfCNCPoint4[5864] = {X 123.7407, Y 19.5139, Z -5.5000, A 0.000, B 0.000, C 0.000 }
gfCNCPoint4[5865] = {X 123.5451, Y 18.1490, Z -5.5000, A 0.000, B 0.000, C 0.000 }
gfCNCPoint4[5866] = {X 123.5444, Y 39.7475, Z -5.5000, A 0.000, B 0.000, C 0.000 }
gfCNCPoint4[5867] = {X 124.1928, Y 40.7414, Z -5.5000, A 0.000, B 0.000, C 0.000 }
gfCNCPoint4[5868] = {X 124.6711, Y 41.8274, Z -5.5000, A 0.000, B 0.000, C 0.000 }
gfCNCPoint4[5869] = {X 124.9666, Y 42.9767, Z -5.5000, A 0.000, B 0.000, C 0.000 }
gfCNCPoint4[5870] = {X 125.0714, Y 44.1587, Z -5.5000, A 0.000, B 0.000, C 0.000 }
gfCNCPoint4[5871] = {X 125.0716, Y 45.0000, Z -5.5000, A 0.000, B 0.000, C 0.000 }
gfCNCPoint4[5872] = {X 124.9610, Y 46.2642, Z -5.5000, A 0.000, B 0.000, C 0.000 }
gfCNCPoint4[5873] = {X 124.6325, Y 47.4899, Z -5.5000, A 0.000, B 0.000, C 0.000 }
gfCNCPoint4[5874] = {X 124.0962, Y 48.6400, Z -5.5000, A 0.000, B 0.000, C 0.000 }
gfCNCPoint4[5875] = {X 123.3684, Y 49.6795, Z -5.5000, A 0.000, B 0.000, C 0.000 }
gfCNCPoint4[5876] = {X 122.4711, Y 50.5768, Z -5.5000, A 0.000, B 0.000, C 0.000 }
gfCNCPoint4[5877] = {X 121.4316, Y 51.3047, Z -5.5000, A 0.000, B 0.000, C 0.000 }
gfCNCPoint4[5878] = {X 120.2815, Y 51.8410, Z -5.5000, A 0.000, B 0.000, C 0.000 }
gfCNCPoint4[5879] = {X 119.0557, Y 52.1694, Z -5.5000, A 0.000, B 0.000, C 0.000 }
gfCNCPoint4[5880] = {X 117.7916, Y 52.2800, Z -5.5000, A 0.000, B 0.000, C 0.000 }
gfCNCPoint4[5881] = {X 111.9185, Y 52.2800, Z -5.5000, A 0.000, B 0.000, C 0.000 }
gfCNCPoint4[5882] = {X 110.8481, Y 52.2009, Z -5.5000, A 0.000, B 0.000, C 0.000 }
gfCNCPoint4[5883] = {X 109.8009, Y 51.9652, Z -5.5000, A 0.000, B 0.000, C 0.000 }
gfCNCPoint4[5884] = {X 108.7998, Y 51.5782, Z -5.5000, A 0.000, B 0.000, C 0.000 }
gfCNCPoint4[5885] = {X 107.8665, Y 51.0481, Z -5.5000, A 0.000, B 0.000, C 0.000 }
gfCNCPoint4[5886] = {X 107.0213, Y 50.3866, Z -5.5000, A 0.000, B 0.000, C 0.000 }
gfCNCPoint4[5887] = {X 106.1743, Y 51.0493, Z -5.5000, A 0.000, B 0.000, C 0.000 }
gfCNCPoint4[5888] = {X 105.2389, Y 51.5800, Z -5.5000, A 0.000, B 0.000, C 0.000 }
gfCNCPoint4[5889] = {X 104.0917, Y 52.0091, Z -5.5000, A 0.000, B 0.000, C 0.000 }
gfCNCPoint4[5890] = {X 102.8887, Y 52.2397, Z -5.5000, A 0.000, B 0.000, C 0.000 }
gfCNCPoint4[5891] = {X 101.6641, Y 52.2655, Z -5.5000, A 0.000, B 0.000, C 0.000 }
gfCNCPoint4[5892] = {X 100.4526, Y 52.0855, Z -5.5000, A 0.000, B 0.000, C 0.000 }
gfCNCPoint4[5893] = {X 99.2883, Y 51.7050, Z -5.5000, A 0.000, B 0.000, C 0.000 }
gfCNCPoint4[5894] = {X 98.2043, Y 51.1347, Z -5.5000, A 0.000, B 0.000, C 0.000 }
gfCNCPoint4[5895] = {X 97.2313, Y 50.3907, Z -5.5000, A 0.000, B 0.000, C 0.000 }
gfCNCPoint4[5896] = {X 96.3865, Y 51.0508, Z -5.5000, A 0.000, B 0.000, C 0.000 }
gfCNCPoint4[5897] = {X 95.4539, Y 51.5797, Z -5.5000, A 0.000, B 0.000, C 0.000 }
gfCNCPoint4[5898] = {X 94.4538, Y 51.9659, Z -5.5000, A 0.000, B 0.000, C 0.000 }
gfCNCPoint4[5899] = {X 93.4078, Y 52.2011, Z -5.5000, A 0.000, B 0.000, C 0.000 }
gfCNCPoint4[5900] = {X 92.3385, Y 52.2800, Z -5.5000, A 0.000, B 0.000, C 0.000 }
gfCNCPoint4[5901] = {X 85.8951, Y 52.2800, Z -5.5000, A 0.000, B 0.000, C 0.000 }
gfCNCPoint4[5902] = {X 84.6852, Y 52.1788, Z -5.5000, A 0.000, B 0.000, C 0.000 }
gfCNCPoint4[5903] = {X 83.5090, Y 51.8779, Z -5.5000, A 0.000, B 0.000, C 0.000 }
gfCNCPoint4[5904] = {X 82.3992, Y 51.3857, Z -5.5000, A 0.000, B 0.000, C 0.000 }
gfCNCPoint4[5905] = {X 81.3866, Y 50.7159, Z -5.5000, A 0.000, B 0.000, C 0.000 }
gfCNCPoint4[5906] = {X 80.5223, Y 52.0937, Z -5.5000, A 0.000, B 0.000, C 0.000 }
gfCNCPoint4[5907] = {X 79.4808, Y 53.3429, Z -5.5000, A 0.000, B 0.000, C 0.000 }
gfCNCPoint4[5908] = {X 78.2809, Y 54.4408, Z -5.5000, A 0.000, B 0.000, C 0.000 }
gfCNCPoint4[5909] = {X 76.9444, Y 55.3676, Z -5.5000, A 0.000, B 0.000, C 0.000 }
gfCNCPoint4[5910] = {X 75.4955, Y 56.1065, Z -5.5000, A 0.000, B 0.000, C 0.000 }
gfCNCPoint4[5911] = {X 73.9605, Y 56.6440, Z -5.5000, A 0.000, B 0.000, C 0.000 }
gfCNCPoint4[5912] = {X 72.3672, Y 56.9705, Z -5.5000, A 0.000, B 0.000, C 0.000 }
gfCNCPoint4[5913] = {X 70.7445, Y 57.0800, Z -5.5000, A 0.000, B 0.000, C 0.000 }
gfCNCPoint4[5914] = {X 64.1851, Y 57.0800, Z -5.5000, A 0.000, B 0.000, C 0.000 }
gfCNCPoint4[5915] = {X 62.6628, Y 56.9837, Z -5.5000, A 0.000, B 0.000, C 0.000 }
gfCNCPoint4[5916] = {X 61.1646, Y 56.6963, Z -5.5000, A 0.000, B 0.000, C 0.000 }
gfCNCPoint4[5917] = {X 59.7147, Y 56.2224, Z -5.5000, A 0.000, B 0.000, C 0.000 }
gfCNCPoint4[5918] = {X 58.3360, Y 55.5695, Z -5.5000, A 0.000, B 0.000, C 0.000 }
gfCNCPoint4[5919] = {X 57.0507, Y 54.7481, Z -5.5000, A 0.000, B 0.000, C 0.000 }
gfCNCPoint4[5920] = {X 55.8790, Y 53.7713, Z -5.5000, A 0.000, B 0.000, C 0.000 }
gfCNCPoint4[5921] = {X 54.7074, Y 54.7481, Z -5.5000, A 0.000, B 0.000, C 0.000 }
gfCNCPoint4[5922] = {X 53.4220, Y 55.5695, Z -5.5000, A 0.000, B 0.000, C 0.000 }
gfCNCPoint4[5923] = {X 52.0434, Y 56.2224, Z -5.5000, A 0.000, B 0.000, C 0.000 }
gfCNCPoint4[5924] = {X 50.5934, Y 56.6963, Z -5.5000, A 0.000, B 0.000, C 0.000 }
gfCNCPoint4[5925] = {X 49.0953, Y 56.9837, Z -5.5000, A 0.000, B 0.000, C 0.000 }
gfCNCPoint4[5926] = {X 47.5729, Y 57.0800, Z -5.5000, A 0.000, B 0.000, C 0.000 }
gfCNCPoint4[5927] = {X 40.6393, Y 57.0800, Z -5.5000, A 0.000, B 0.000, C 0.000 }
gfCNCPoint4[5928] = {X 39.3238, Y 57.0082, Z -5.5000, A 0.000, B 0.000, C 0.000 }
gfCNCPoint4[5929] = {X 38.0239, Y 56.7935, Z -5.5000, A 0.000, B 0.000, C 0.000 }
gfCNCPoint4[5930] = {X 36.7552, Y 56.4385, Z -5.5000, A 0.000, B 0.000, C 0.000 }
gfCNCPoint4[5931] = {X 35.5327, Y 55.9475, Z -5.5000, A 0.000, B 0.000, C 0.000 }
gfCNCPoint4[5932] = {X 34.1216, Y 56.7826, Z -5.5000, A 0.000, B 0.000, C 0.000 }
gfCNCPoint4[5933] = {X 32.6344, Y 57.4726, Z -5.5000, A 0.000, B 0.000, C 0.000 }
gfCNCPoint4[5934] = {X 31.0857, Y 58.0109, Z -5.5000, A 0.000, B 0.000, C 0.000 }
gfCNCPoint4[5935] = {X 29.4910, Y 58.3919, Z -5.5000, A 0.000, B 0.000, C 0.000 }
gfCNCPoint4[5936] = {X 27.8662, Y 58.6120, Z -5.5000, A 0.000, B 0.000, C 0.000 }
gfCNCPoint4[5937] = {X 25.6546, Y 59.5467, Z -5.5000, A 0.000, B 0.000, C 0.000 }
gfCNCPoint4[5938] = {X 23.3924, Y 60.3513, Z -5.5000, A 0.000, B 0.000, C 0.000 }
gfCNCPoint4[5939] = {X 21.1517, Y 61.0065, Z -5.5000, A 0.000, B 0.000, C 0.000 }
gfCNCPoint4[5940] = {X 18.8721, Y 61.5102, Z -5.5000, A 0.000, B 0.000, C 0.000 }
gfCNCPoint4[5941] = {X 16.5640, Y 61.8602, Z -5.5000, A 0.000, B 0.000, C 0.000 }
gfCNCPoint4[5942] = {X 14.2376, Y 62.0548, Z -5.5000, A 0.000, B 0.000, C 0.000 }
gfCNCPoint4[5943] = {X 11.9034, Y 62.0932, Z -5.5000, A 0.000, B 0.000, C 0.000 }
gfCNCPoint4[5944] = {X 11.9034, Y 88.0951, Z -5.5000, A 0.000, B 0.000, C 0.000 }
gfCNCPoint4[5945] = {X 113.6324, Y 88.0951, Z -5.5000, A 0.000, B 0.000, C 0.000 }
gfCNCPoint4[5946] = {X 114.7659, Y 86.8202, Z -5.5000, A 0.000, B 0.000, C 0.000 }
gfCNCPoint4[5947] = {X 116.0415, Y 85.6874, Z -5.5000, A 0.000, B 0.000, C 0.000 }
gfCNCPoint4[5948] = {X 117.4414, Y 84.7126, Z -5.5000, A 0.000, B 0.000, C 0.000 }
gfCNCPoint4[5949] = {X 118.9463, Y 83.9091, Z -5.5000, A 0.000, B 0.000, C 0.000 }
gfCNCPoint4[5950] = {X 120.5352, Y 83.2882, Z -5.5000, A 0.000, B 0.000, C 0.000 }
gfCNCPoint4[5951] = {X 122.1861, Y 82.8585, Z -5.5000, A 0.000, B 0.000, C 0.000 }
gfCNCPoint4[5952] = {X 144.8180, Y 58.0055, Z -5.5000, A 0.000, B 0.000, C 0.000 }
gfCNCPoint4[5953] = {X 144.9144, Y 56.3315, Z -5.5000, A 0.000, B 0.000, C 0.000 }
gfCNCPoint4[5954] = {X 145.2037, Y 54.6800, Z -5.5000, A 0.000, B 0.000, C 0.000 }
gfCNCPoint4[5955] = {X 143.0396, Y 54.6800, Z -5.5000, A 0.000, B 0.000, C 0.000 }
gfCNCPoint4[5956] = {X 142.7948, Y 54.6769, Z -5.5000, A 0.000, B 0.000, C 0.000 }
gfCNCPoint4[5957] = {X 142.5501, Y 54.6676, Z -5.5000, A 0.000, B 0.000, C 0.000 }
gfCNCPoint4[5958] = {X 141.0972, Y 54.4831, Z -5.5000, A 0.000, B 0.000, C 0.000 }
gfCNCPoint4[5959] = {X 139.6887, Y 54.0815, Z -5.5000, A 0.000, B 0.000, C 0.000 }
gfCNCPoint4[5960] = {X 138.3569, Y 53.4720, Z -5.5000, A 0.000, B 0.000, C 0.000 }
gfCNCPoint4[5961] = {X 137.1323, Y 52.6685, Z -5.5000, A 0.000, B 0.000, C 0.000 }
gfCNCPoint4[5962] = {X 136.0429, Y 51.6895, Z -5.5000, A 0.000, B 0.000, C 0.000 }
gfCNCPoint4[5963] = {X 135.1138, Y 50.5573, Z -5.5000, A 0.000, B 0.000, C 0.000 }
gfCNCPoint4[5964] = {X 134.3661, Y 49.2979, Z -5.5000, A 0.000, B 0.000, C 0.000 }
gfCNCPoint4[5965] = {X 133.8169, Y 47.9401, Z -5.5000, A 0.000, B 0.000, C 0.000 }
gfCNCPoint4[5966] = {X 133.4789, Y 46.5150, Z -5.5000, A 0.000, B 0.000, C 0.000 }
gfCNCPoint4[5967] = {X 133.3598, Y 45.0552, Z -5.5000, A 0.000, B 0.000, C 0.000 }
gfCNCPoint4[5968] = {X 133.3601, Y 44.1105, Z -5.5000, A 0.000, B 0.000, C 0.000 }
gfCNCPoint4[5969] = {X 133.4665, Y 42.7743, Z -5.5000, A 0.000, B 0.000, C 0.000 }
gfCNCPoint4[5970] = {X 133.7565, Y 41.4655, Z -5.5000, A 0.000, B 0.000, C 0.000 }
gfCNCPoint4[5971] = {X 136.0581, Y 42.1457, Z -5.5000, A 0.000, B 0.000, C 0.000 }
gfCNCPoint4[5972] = {X 136.3664, Y 41.2990, Z -5.5000, A 0.000, B 0.000, C 0.000 }
gfCNCPoint4[5973] = {X 136.7770, Y 40.4969, Z -5.5000, A 0.000, B 0.000, C 0.000 }
gfCNCPoint4[5974] = {X 137.2836, Y 39.7516, Z -5.5000, A 0.000, B 0.000, C 0.000 }
gfCNCPoint4[5975] = {X 137.2836, Y 23.8768, Z -5.5000, A 0.000, B 0.000, C 0.000 }
gfCNCPoint4[5976] = {X 136.4352, Y 24.2641, Z -5.5000, A 0.000, B 0.000, C 0.000 }
gfCNCPoint4[5977] = {X 135.5443, Y 24.5398, Z -5.5000, A 0.000, B 0.000, C 0.000 }
gfCNCPoint4[5978] = {X 134.6254, Y 24.6993, Z -5.5000, A 0.000, B 0.000, C 0.000 }
gfCNCPoint4[5979] = {X 134.2595, Y 24.7296, Z -5.5000, A 0.000, B 0.000, C 0.000 }
gfCNCPoint4[5980] = {X 133.8926, Y 24.7414, Z -5.5000, A 0.000, B 0.000, C 0.000 }
gfCNCPoint4[5981] = {X 133.2006, Y 24.7415, Z -5.5000, A 0.000, B 0.000, C 0.000 }
gfCNCPoint4[5982] = {X 131.9931, Y 24.6407, Z -5.5000, A 0.000, B 0.000, C 0.000 }
gfCNCPoint4[5983] = {X 130.8191, Y 24.3410, Z -5.5000, A 0.000, B 0.000, C 0.000 }
gfCNCPoint4[5984] = {X 129.7110, Y 23.8507, Z -5.5000, A 0.000, B 0.000, C 0.000 }
gfCNCPoint4[5985] = {X 128.6996, Y 23.1834, Z -5.5000, A 0.000, B 0.000, C 0.000 }
gfCNCPoint4[5986] = {X 127.8129, Y 22.3575, Z -5.5000, A 0.000, B 0.000, C 0.000 }
gfCNCPoint4[5987] = {X 127.0755, Y 21.3961, Z -5.5000, A 0.000, B 0.000, C 0.000 }
gfCNCPoint4[5988] = {X 126.5077, Y 20.3256, Z -5.5000, A 0.000, B 0.000, C 0.000 }
gfCNCPoint4[5989] = {X 126.1254, Y 19.1758, Z -5.5000, A 0.000, B 0.000, C 0.000 }
gfCNCPoint4[5990] = {X 125.9390, Y 17.9785, Z -5.5000, A 0.000, B 0.000, C 0.000 }
gfCNCPoint4[5991] = {X 125.9252, Y 17.7202, Z -5.5000, A 0.000, B 0.000, C 0.000 }
gfCNCPoint4[5992] = {X 125.9206, Y 17.4615, Z -5.5000, A 0.000, B 0.000, C 0.000 }
gfCNCPoint4[5993] = {X 125.9206, Y 10.4835, Z -5.5000, A 0.000, B 0.000, C 0.000 }
gfCNCPoint4[5994] = {X 125.9372, Y 9.9931, Z -5.5000, A 0.000, B 0.000, C 0.000 }
gfCNCPoint4[5995] = {X 125.9867, Y 9.5049, Z -5.5000, A 0.000, B 0.000, C 0.000 }
gfCNCPoint4[5996] = {X 121.8686, Y 9.5049, Z -5.5000, A 0.000, B 0.000, C 0.000 }
gfCNCPoint4[5997] = {X 122.3090, Y 10.3410, Z -5.5000, A 0.000, B 0.000, C 0.000 }
gfCNCPoint4[5998] = {X 122.5801, Y 11.2463, Z -5.5000, A 0.000, B 0.000, C 0.000 }
gfCNCPoint4[5999] = {X 122.6716, Y 12.1868, Z -5.5000, A 0.000, B 0.000, C 0.000 }
gfCNCPoint4[6000] = {X 122.6714, Y 13.0237, Z -5.5000, A 0.000, B 0.000, C 0.000 }
gfCNCPoint4[6001] = {X 122.5640, Y 13.9968, Z -5.5000, A 0.000, B 0.000, C 0.000 }
gfCNCPoint4[6002] = {X 122.2647, Y 14.9289, Z -5.5000, A 0.000, B 0.000, C 0.000 }
gfCNCPoint4[6003] = {X 121.7853, Y 15.7825, Z -5.5000, A 0.000, B 0.000, C 0.000 }
gfCNCPoint4[6004] = {X 121.1451, Y 16.5232, Z -5.5000, A 0.000, B 0.000, C 0.000 }
gfCNCPoint4[6005] = {X 121.1444, Y 40.6629, Z -5.5000, A 0.000, B 0.000, C 0.000 }
gfCNCPoint4[6006] = {X 121.7856, Y 41.4049, Z -5.5000, A 0.000, B 0.000, C 0.000 }
gfCNCPoint4[6007] = {X 122.2656, Y 42.2601, Z -5.5000, A 0.000, B 0.000, C 0.000 }
gfCNCPoint4[6008] = {X 122.5649, Y 43.1939, Z -5.5000, A 0.000, B 0.000, C 0.000 }
gfCNCPoint4[6009] = {X 122.6714, Y 44.1688, Z -5.5000, A 0.000, B 0.000, C 0.000 }
gfCNCPoint4[6010] = {X 122.6716, Y 45.0000, Z -5.5000, A 0.000, B 0.000, C 0.000 }
gfCNCPoint4[6011] = {X 122.5778, Y 45.9520, Z -5.5000, A 0.000, B 0.000, C 0.000 }
gfCNCPoint4[6012] = {X 122.3001, Y 46.8675, Z -5.5000, A 0.000, B 0.000, C 0.000 }
gfCNCPoint4[6013] = {X 121.8491, Y 47.7112, Z -5.5000, A 0.000, B 0.000, C 0.000 }
gfCNCPoint4[6014] = {X 121.2423, Y 48.4507, Z -5.5000, A 0.000, B 0.000, C 0.000 }
gfCNCPoint4[6015] = {X 120.5028, Y 49.0576, Z -5.5000, A 0.000, B 0.000, C 0.000 }
gfCNCPoint4[6016] = {X 119.6591, Y 49.5085, Z -5.5000, A 0.000, B 0.000, C 0.000 }
gfCNCPoint4[6017] = {X 118.7436, Y 49.7862, Z -5.5000, A 0.000, B 0.000, C 0.000 }
gfCNCPoint4[6018] = {X 117.7916, Y 49.8800, Z -5.5000, A 0.000, B 0.000, C 0.000 }
gfCNCPoint4[6019] = {X 111.9185, Y 49.8800, Z -5.5000, A 0.000, B 0.000, C 0.000 }
gfCNCPoint4[6020] = {X 111.0234, Y 49.7972, Z -5.5000, A 0.000, B 0.000, C 0.000 }
gfCNCPoint4[6021] = {X 110.1587, Y 49.5517, Z -5.5000, A 0.000, B 0.000, C 0.000 }
gfCNCPoint4[6022] = {X 109.3537, Y 49.1517, Z -5.5000, A 0.000, B 0.000, C 0.000 }
gfCNCPoint4[6023] = {X 108.6357, Y 48.6108, Z -5.5000, A 0.000, B 0.000, C 0.000 }
gfCNCPoint4[6024] = {X 108.0714, Y 48.0024, Z -5.5000, A 0.000, B 0.000, C 0.000 }
gfCNCPoint4[6025] = {X 107.6183, Y 47.3071, Z -5.5000, A 0.000, B 0.000, C 0.000 }
gfCNCPoint4[6026] = {X 107.2895, Y 46.5451, Z -5.5000, A 0.000, B 0.000, C 0.000 }
gfCNCPoint4[6027] = {X 107.0947, Y 45.7384, Z -5.5000, A 0.000, B 0.000, C 0.000 }
gfCNCPoint4[6028] = {X 106.6287, Y 46.8769, Z -5.5000, A 0.000, B 0.000, C 0.000 }
gfCNCPoint4[6029] = {X 106.1131, Y 47.8111, Z -5.5000, A 0.000, B 0.000, C 0.000 }
gfCNCPoint4[6030] = {X 105.4068, Y 48.6108, Z -5.5000, A 0.000, B 0.000, C 0.000 }
gfCNCPoint4[6031] = {X 104.8391, Y 49.0550, Z -5.5000, A 0.000, B 0.000, C 0.000 }
gfCNCPoint4[6032] = {X 104.2121, Y 49.4107, Z -5.5000, A 0.000, B 0.000, C 0.000 }
gfCNCPoint4[6033] = {X 103.3106, Y 49.7335, Z -5.5000, A 0.000, B 0.000, C 0.000 }
gfCNCPoint4[6034] = {X 102.3635, Y 49.8741, Z -5.5000, A 0.000, B 0.000, C 0.000 }
gfCNCPoint4[6035] = {X 101.4071, Y 49.8271, Z -5.5000, A 0.000, B 0.000, C 0.000 }
gfCNCPoint4[6036] = {X 100.4784, Y 49.5941, Z -5.5000, A 0.000, B 0.000, C 0.000 }
gfCNCPoint4[6037] = {X 99.6130, Y 49.1844, Z -5.5000, A 0.000, B 0.000, C 0.000 }
gfCNCPoint4[6038] = {X 98.8443, Y 48.6135, Z -5.5000, A 0.000, B 0.000, C 0.000 }
gfCNCPoint4[6039] = {X 98.1362, Y 47.8127, Z -5.5000, A 0.000, B 0.000, C 0.000 }
gfCNCPoint4[6040] = {X 97.6194, Y 46.8769, Z -5.5000, A 0.000, B 0.000, C 0.000 }
gfCNCPoint4[6041] = {X 97.1600, Y 45.7536, Z -5.5000, A 0.000, B 0.000, C 0.000 }
gfCNCPoint4[6042] = {X 96.9635, Y 46.5570, Z -5.5000, A 0.000, B 0.000, C 0.000 }
gfCNCPoint4[6043] = {X 96.6342, Y 47.3156, Z -5.5000, A 0.000, B 0.000, C 0.000 }
gfCNCPoint4[6044] = {X 96.1814, Y 48.0078, Z -5.5000, A 0.000, B 0.000, C 0.000 }
gfCNCPoint4[6045] = {X 95.6183, Y 48.6135, Z -5.5000, A 0.000, B 0.000, C 0.000 }
gfCNCPoint4[6046] = {X 94.9007, Y 49.1533, Z -5.5000, A 0.000, B 0.000, C 0.000 }
gfCNCPoint4[6047] = {X 94.0964, Y 49.5524, Z -5.5000, A 0.000, B 0.000, C 0.000 }
gfCNCPoint4[6048] = {X 93.2326, Y 49.7974, Z -5.5000, A 0.000, B 0.000, C 0.000 }
gfCNCPoint4[6049] = {X 92.3385, Y 49.8800, Z -5.5000, A 0.000, B 0.000, C 0.000 }
gfCNCPoint4[6050] = {X 85.8951, Y 49.8800, Z -5.5000, A 0.000, B 0.000, C 0.000 }
gfCNCPoint4[6051] = {X 85.0841, Y 49.8121, Z -5.5000, A 0.000, B 0.000, C 0.000 }
gfCNCPoint4[6052] = {X 84.2956, Y 49.6104, Z -5.5000, A 0.000, B 0.000, C 0.000 }
gfCNCPoint4[6053] = {X 83.5517, Y 49.2805, Z -5.5000, A 0.000, B 0.000, C 0.000 }
gfCNCPoint4[6054] = {X 82.8729, Y 48.8316, Z -5.5000, A 0.000, B 0.000, C 0.000 }
